F_CALC_SENSOR_POS( N44_AI2_CH5_4 * 0.004, ALARMS.Clear, LS301 );
F_CALC_SENSOR_POS( N44_AI0_CH6_4 * 0.004, ALARMS.Clear, LS303 );
F_CALC_SENSOR_POS( N44_AI4_CH8_4 * 0.004, ALARMS.Clear, LS305 );

F_CALC_SENSOR_KG( P301.Bar, L301 );
F_CALC_SENSOR_KG( P303.Bar, L303 );
F_CALC_SENSOR_KG( P305.Bar, L305 );
F_CALC_SENSOR_KG( P307.Bar, L307 );
F_CALC_SENSOR_KG( P309.Bar, L309 );
F_CALC_SENSOR_KG( P311.Bar, L311 );

(*MF04 - Node44*)
SF402 := N38_DI7_CH8_2;
SF403 := N38_DI6_CH8_4;
SF404 := N44_DI1_CH7_2;
SF405 := N44_DI0_CH7_4;

(*MF05 - Node41*)
F_CALC_SENSOR_BAR( N41_AI3_CH5_2 * 0.004, ALARMS.Clear,  P501 );
F_CALC_SENSOR_BAR( N41_AI2_CH5_4 * 0.004, ALARMS.Clear,  P503 );
F_CALC_SENSOR_BAR( N41_AI1_CH6_2 * 0.004, ALARMS.Clear,  P507 );
F_CALC_SENSOR_BAR( N41_AI0_CH6_4 * 0.004, ALARMS.Clear,  P505 );

(*F_CALC_SENSOR_KG( P501.Bar, L501 );*)
F_CALC_SENSOR_KG( P503.Bar, L503 );
F_CALC_SENSOR_KG( P505.Bar, L505 );
L501_7 := P501.Bar * L501.Cal_K - P507.Bar * L501.Cal_C;

(*MF06 - Node20/47*)
F_CALC_SENSOR_BAR ( N20_AI3_CH5_2 * 0.004, ALARMS.Clear,  P601 );
F_CALC_SENSOR_BAR ( N20_AI2_CH5_4 * 0.004, ALARMS.Clear,  P603 );
F_CALC_SENSOR_BAR ( N20_AI1_CH6_2 * 0.004, ALARMS.Clear,  P605 );
F_CALC_SENSOR_BAR ( N20_AI0_CH6_4 * 0.004, ALARMS.Clear,  P607 );

F_CALC_SENSOR_POS ( N47_AI1_CH6_2 * 0.004, ALARMS.Clear, LS601 );
F_CALC_SENSOR_POS ( N20_AI4_CH8_4 * 0.004, ALARMS.Clear, LS605 );


(*MF07 - Node21/22*)
F_CALC_SENSOR_BAR( N21_AI3_CH5_2 * 0.004, ALARMS.Clear,  P701 );
F_CALC_SENSOR_BAR( N21_AI2_CH5_4 * 0.004, ALARMS.Clear,  P703 );

F_CALC_SENSOR_POS( N21_AI1_CH6_2 * 0.004, ALARMS.Clear, LS707 );
F_CALC_SENSOR_POS( N21_AI0_CH6_4 * 0.004, ALARMS.Clear, LS709 );

F_CALC_SENSOR_BAR( N22_AI3_CH5_2 * 0.004, ALARMS.Clear,  P707 );
F_CALC_SENSOR_BAR( N22_AI2_CH5_4 * 0.004, ALARMS.Clear,  P709 );
F_CALC_SENSOR_BAR( N22_AI1_CH6_2 * 0.004, ALARMS.Clear,  P705 );

F_CALC_SENSOR_KG( P701.Bar, L701 );
F_CALC_SENSOR_KG( P703.Bar, L703 );
F_CALC_SENSOR_KG( P705.Bar, L705 );
F_CALC_SENSOR_KG( P707.Bar, L707 );
F_CALC_SENSOR_KG( P709.Bar, L709 );

(*MF08 - Node23*)
F_CALC_SENSOR_NC ( NOT N39_DI3_CH6_2 , ALARMS.Clear, MAIN.Cycle_Time, 0.0, SF801 );
F_CALC_SENSOR_NC ( NOT N39_DI2_CH6_4 , ALARMS.Clear, MAIN.Cycle_Time, 0.0, SF803 );

F_CALC_SENSOR_BAR( N23_AI1_CH6_2 * 0.004, ALARMS.Clear,  P804 );(**)
F_CALC_SENSOR_BAR( N23_AI0_CH6_4 * 0.004, ALARMS.Clear,  P802 );(**)

F_CALC_SENSOR_POS( N23_AI3_CH5_2 * 0.004, ALARMS.Clear, LS803 );(**)
F_CALC_SENSOR_POS( N23_AI2_CH5_4 * 0.004, ALARMS.Clear, LS801 );(**)

(*MF09 - Node35*)
F_CALC_SENSOR_BAR( N35_AI3_CH5_2 * 0.004, ALARMS.Clear,  P901 );
F_CALC_SENSOR_BAR( N35_AI2_CH5_4 * 0.004, ALARMS.Clear,  P903 );
F_CALC_SENSOR_BAR( N35_AI1_CH6_2 * 0.004, ALARMS.Clear,  P905 );
F_CALC_SENSOR_BAR( N35_AI0_CH6_4 * 0.004, ALARMS.Clear,  P907 );

F_CALC_SENSOR_KG( P901.Bar, L901 );
F_CALC_SENSOR_KG( P903.Bar, L903 );

F_CALC_SENSOR_POS( N38_AI3_CH5_2 * 0.004, ALARMS.Clear, LS901 );
F_CALC_SENSOR_POS( N38_AI2_CH5_4 * 0.004, ALARMS.Clear, LS903 );

(*MF10 - Node39/40*)
F_CALC_SENSOR_NC ( N39_DI1_CH7_2, ALARMS.Clear, MAIN.Cycle_Time, 0.0            , SF1002 );
F_CALC_SENSOR_NC (NOT N40_DI7_CH8_2, ALARMS.Clear, MAIN.Cycle_Time, PARAMS.SF_Delay, SF1003 );
F_CALC_SENSOR_NC (NOT N40_DI6_CH8_4, ALARMS.Clear, MAIN.Cycle_Time, PARAMS.SF_Delay, SF1004 );

F_CALC_SENSOR_BAR( N40_AI3_CH5_2 * 0.004, ALARMS.Clear,  P1001 );
F_CALC_SENSOR_BAR( N40_AI2_CH5_4 * 0.004, ALARMS.Clear,  P1002 );
F_CALC_SENSOR_POS( N40_AI1_CH6_2 * 0.004, ALARMS.Clear, LS1002 );(**)
F_CALC_SENSOR_POS( N40_AI0_CH6_4 * 0.004, ALARMS.Clear, LS1001 );(**)

(*MF11 - Node47*)
F_CALC_SENSOR_BAR( N47_AI3_CH5_2 * 0.004, ALARMS.Clear,  P1101 );
F_CALC_SENSOR_BAR( N47_AI2_CH5_4 * 0.004, ALARMS.Clear,  P1102 );

F_CALC_SENSOR_TEMP( N47_AI4_CH8_4 * 0.001, ALARMS.Clear, MAIN.Cycle_Time, S1100 );

(*MF12 - Node24/25*)
F_CALC_SENSOR_BAR( N24_AI7_CH3_2 * 0.001, ALARMS.Clear,  P1216 );
F_CALC_SENSOR_BAR( N24_AI6_CH3_4 * 0.001, ALARMS.Clear,  P1219 );
F_CALC_SENSOR_BAR( N24_AI3_CH5_2 * 0.001, ALARMS.Clear,  P1214 );
F_CALC_SENSOR_BAR( N24_AI2_CH5_4 * 0.001, ALARMS.Clear,  P1215 );
F_CALC_SENSOR_BAR( N24_AI1_CH6_2 * 0.001, ALARMS.Clear,  P1212 );
F_CALC_SENSOR_BAR( N24_AI0_CH6_4 * 0.001, ALARMS.Clear,  P1213 );
F_CALC_SENSOR_BAR( N24_AI5_CH8_2 * 0.001, ALARMS.Clear,  P1210 );
F_CALC_SENSOR_BAR( N24_AI4_CH8_4 * 0.001, ALARMS.Clear,  P1211 );

F_CALC_SENSOR_BAR( N25_AI7_CH3_2 * 0.001, ALARMS.Clear,  P1208 );
F_CALC_SENSOR_BAR( N25_AI6_CH3_4 * 0.001, ALARMS.Clear,  P1209 );
F_CALC_SENSOR_BAR( N25_AI3_CH5_2 * 0.001, ALARMS.Clear,  P1206 );
F_CALC_SENSOR_BAR( N25_AI2_CH5_4 * 0.001, ALARMS.Clear,  P1207 );
F_CALC_SENSOR_BAR( N25_AI1_CH6_2 * 0.001, ALARMS.Clear,  P1204 );
F_CALC_SENSOR_BAR( N25_AI0_CH6_4 * 0.001, ALARMS.Clear,  P1205 );
F_CALC_SENSOR_BAR( N25_AI5_CH8_2 * 0.001, ALARMS.Clear,  P1202 );
F_CALC_SENSOR_BAR( N25_AI4_CH8_4 * 0.001, ALARMS.Clear,  P1203 );

(*MF13 - Node33 - Traveller*)
SF1301 := N38_DI1_CH7_2;
SF1302 := N38_DI0_CH7_4;

F_CALC_SENSOR_BAR( N33_AI3_CH5_2 * 0.004, ALARMS.Clear,  P1302 );
F_CALC_SENSOR_BAR( N33_AI2_CH5_4 * 0.004, ALARMS.Clear,  P1301 );

F_CALC_SENSOR_POS( N38_AI1_CH6_2 * 0.004, ALARMS.Clear, LS1303 );

(*MF16 - Node34*)
F_CALC_SENSOR_BAR( N34_AI3_CH5_2 * 0.001, ALARMS.Clear,  P1603 );
F_CALC_SENSOR_BAR( N34_AI2_CH5_4 * 0.001, ALARMS.Clear,  P1605 );
F_CALC_SENSOR_BAR( N34_AI1_CH6_2 * 0.001, ALARMS.Clear,  P1604 );
F_CALC_SENSOR_BAR( N34_AI0_CH6_4 * 0.001, ALARMS.Clear,  P1602 );

(*MF19 - Node32*)
F_CALC_SENSOR_POS( N32_AI1_CH6_2 * 0.004, ALARMS.Clear, LS1905 );

SF1909 := N32_DI1_CH7_2;
SF1911 := N32_DI0_CH7_4;
SF1901 := N32_DI7_CH8_2;
SF1903 := N32_DI6_CH8_4;

(*MF20 - Node31*)
F_CALC_SENSOR_POS( N31_AI3_CH5_2 * 0.004, ALARMS.Clear, LS2001 );
F_CALC_SENSOR_POS( N31_AI2_CH5_4 * 0.001, ALARMS.Clear, LS2005 );

SF2009 := N31_DI1_CH7_2;
SF2011 := N31_DI0_CH7_4;

(*MF21 - Node28*)
SF2101 := N28_DI5_CH5_2;
SF2103 := N28_DI4_CH5_4;
SF2105 := N28_DI3_CH6_2;
SF2107 := N28_DI2_CH6_4;
SF2109 := N28_DI1_CH7_2;
SF2111 := N28_DI0_CH7_4;

(*MF22 - Node27*)
SF2205 := N27_DI3_CH6_2;
SF2207 := N27_DI2_CH6_4;
SF2209 := N27_DI1_CH7_2;
SF2211 := N27_DI0_CH7_4;

(*MF23 - Node30*)
F_CALC_SENSOR_POS( N30_AI3_CH5_2 * 0.004, ALARMS.Clear, LS021  );
F_CALC_SENSOR_POS( N30_AI2_CH5_4 * 0.004, ALARMS.Clear, LS022  );
F_CALC_SENSOR_POS( N30_AI1_CH6_2 * 0.004, ALARMS.Clear, LS2301 );
F_CALC_SENSOR_POS( N30_AI0_CH6_4 * 0.004, ALARMS.Clear, LS2305 );

SF2309 := N30_DI1_CH7_2;
SF2311 := N30_DI0_CH7_4;
SF021  := N30_DI7_CH8_2;
SF022  := N30_DI6_CH8_4;

(*MF24 - Node29*)
F_CALC_SENSOR_POS( N29_AI3_CH5_2 * 0.001, ALARMS.Clear, LS2401 );
F_CALC_SENSOR_POS( N29_AI2_CH5_4 * 0.004, ALARMS.Clear, LS2409 );
F_CALC_SENSOR_POS( N29_AI1_CH6_2 * 0.004, ALARMS.Clear, LS2201 );
F_CALC_SENSOR_POS( N29_AI0_CH6_4 * 0.004, ALARMS.Clear, LS023  );

SF2405 := N29_DI1_CH7_2;
SF2407 := N29_DI0_CH7_4;

(*MF25 - Node26*)
F_CALC_SENSOR_POS( N26_AI3_CH5_2 * 0.004, ALARMS.Clear, LS2501 );
F_CALC_SENSOR_POS( N26_AI2_CH5_4 * 0.004, ALARMS.Clear, LS2505 );
F_CALC_SENSOR_BAR( N26_AI1_CH6_2 * 0.004, ALARMS.Clear, P2500  );
F_CALC_SENSOR_POS( N26_AI0_CH6_4 * 0.004, ALARMS.Clear, LS024  );

SF023  := N26_DI7_CH8_2;
SF024  := N26_DI6_CH8_4;


(*DGB Sela - Node48*)
F_CALC_SENSOR_BAR ( N48_AI3_CH5_2 * 0.004, ALARMS.Clear,  P_SealP );
F_CALC_SENSOR_BAR ( N48_AI1_CH6_2 * 0.004, ALARMS.Clear,  P_SealS );


(*L102_raw := P102_bar * PARAMS.stL102_Cal.K;*)

(*L102_Kg := L102_raw * (PARAMS.stL102_Cal.C / 100.0);*)

(*Buttons*)
(*FRO TACK*)
B301[1] := N102_IN.2;
B302[1] := N102_IN.3;
B301[2] := N113_IN.3;
B302[2] := N113_IN.2;
(*A3 TACK*)
B303[1] := N102_IN.4;
B304[1] := N102_IN.5;
B303[2] := N113_IN.5;
B304[2] := N113_IN.4;
(*J5*)
B305[1] := N118_IN.6;
B306[1] := N118_IN.7;
B305[2] := N119_IN.7;
B306[2] := N119_IN.6;
(*J4*)
B307[1] := N118_IN.8;
B308[1] := N118_IN.9;
B307[2] := N119_IN.9;
B308[2] := N119_IN.8;
(*FORESTAY*)
B309[1] := N104_IN.1;
B310[1] := N104_IN.0;
B309[2] := N105_IN.0;
B310[2] := N105_IN.1;
(*J2*)
B311[1] := N114_IN.4;
B312[1] := N114_IN.5;
B311[2] := N115_IN.5;
B312[2] := N115_IN.4;
(*JIB INOUT*)
B501[1] := N114_IN.2;
B502[1] := N114_IN.3;
B501[2] := N115_IN.3;
B502[2] := N115_IN.2;
(*JIB UPDW*)
B503[1] := N114_IN.0;
B504[1] := N114_IN.1;
B503[2] := N115_IN.1;
B504[2] := N115_IN.0;
(*VANG*)
(*B505 [1] := N116_IN.4;
B506 [1] := N116_IN.5;
B506Q[1] := N116_IN.5 AND N116_IN.0;
B505 [2] := N117_IN.5;
B506 [2] := N117_IN.4;
B506Q[2] := N117_IN.4 AND N117_IN.1;*)

(*PORP UP/DW*)
B601[1] := N112_IN.3; (*DW*)
B603[1] := N112_IN.2; (*UP*)
(*TRIM TAB*)
B605[1] := N104_IN.3;
B607[1] := N104_IN.2;
B606[1] := N104_IN.4;
B605[2] := N105_IN.3;
B607[2] := N105_IN.2;
B606[2] := N105_IN.5;

(*INNER STAYSAIL*)
B701[1] := N102_IN.0;
B702[1] := N102_IN.1;
B701[2] := N113_IN.1;
B702[2] := N113_IN.0;
(*MAIN OUTHAUL*)
B703[1] := N116_IN.8;
B704[1] := N116_IN.9;
B703[2] := N117_IN.9;
B704[2] := N117_IN.8;
(*MAIN CUNNINGHAM*)
B705[1] := N116_IN.6;
B706[1] := N116_IN.7;
B705[2] := N117_IN.7;
B706[2] := N117_IN.6;
(*BOTTOM DEFLECTOR*)
B707[1] := N118_IN.2;
B708[1] := N118_IN.3;
B707[2] := N119_IN.3;
B708[2] := N119_IN.2;
(*TOP DEFLECTOR*)
B709[1] := N118_IN.4;
B710[1] := N118_IN.5;
B709[2] := N119_IN.5;
B710[2] := N119_IN.4;

(*BACSTAY PORT*)
(*B901[1] := N104_IN.7; (*Panel Stbd works on Backstay Port*)
B902[1] := N104_IN.6;

B901[2] := N118_IN.0; (*Panel Port works on Backstay Port Fine Tune*)
B902[2] := N118_IN.1;*)

(*BACKSTAY STBD*)
(*B903[1] := N105_IN.6; (*Panel Port works on Backstay Stbd*)
B904[1] := N105_IN.7;

B903[2] := N119_IN.1; (*Panel Stbd works on Backstay Stbd Fine Tune*)
B904[2] := N119_IN.0;*)

(*BACKSTAY TACK*)
(*B90T[1] := N104_IN.5;
B90T[2] := N105_IN.4;*)
(******************************************************fine tune y TACK***)

(*TRAVELLER*)
BTravA[1] := N116_IN.3;
BTravB[1] := N116_IN.2;
BTravT[1] := N116_IN.1;
BTravD[1] := N116_IN.1 AND N116_IN.0;

BTravA[2] := N117_IN.3;
BTravB[2] := N117_IN.2;
BTravT[2] := N117_IN.0;
BTravD[2] := N117_IN.0 AND N117_IN.1;

BTravA[3] := N38_DI0_CH7_4; (******************************Verificar cual es Port y Stbd***)
BTravB[3] := N38_DI1_CH7_2;

(*KEEL*)
BKeelP[1] := N110_IN.0;
BKeelS[1] := N110_IN.4;
BKeelC[1] := N110_IN.3;
BKeelF[1] := N110_IN.2;
BKeelT[1] := N110_IN.5;

BKeelP[2] := N111_IN.0;
BKeelS[2] := N111_IN.4;
BKeelC[2] := N111_IN.3;
BKeelF[2] := N111_IN.2;
BKeelT[2] := N111_IN.5;

(*BKeelP[3] := N108_IN.0;
BKeelS[3] := N108_IN.4;
BKeelC[3] := N108_IN.3;
BKeelF[3] := N108_IN.2;

BKeelP[4] := N109_IN.0;
BKeelS[4] := N109_IN.4;
BKeelC[4] := N109_IN.3;
BKeelF[4] := N109_IN.2;*) (*Now Mast setup*)

(*BOARD*)
BBoardP[1] := MAIN.fbMastSetup.State_MS = 0 AND N108_IN.6;
BBoardS[1] := MAIN.fbMastSetup.State_MS = 0 AND N108_IN.7;
BBoardC[1] := MAIN.fbMastSetup.State_MS = 0 AND N108_IN.5;

BBoardP[2] := MAIN.fbMastSetup.State_HS = 0 AND N109_IN.6;
BBoardS[2] := MAIN.fbMastSetup.State_HS = 0 AND N109_IN.7;
BBoardC[2] := MAIN.fbMastSetup.State_HS = 0 AND N109_IN.5;

(*Bow Thruster*)
BBowThrP := N38_DI7_CH8_2;
BBowThrS := N38_DI6_CH8_4;
BBowThrU := N112_IN.4;
BBowThrD := N112_IN.5;

(*Water Ballast*)
BWB_P_Fwd[1] := N106_IN.0;
BWB_S_Fwd[1] := N106_IN.1;
BWB_P_Aft[1] := N106_IN.2;
BWB_S_Aft[1] := N106_IN.3;
BWB_Fill [1] := N106_IN.4;
BWB_Dump [1] := N106_IN.5;
BWB_Stop [1] := N106_IN.7;
BWB_12   [1] := N106_IN.8;
BWB_Move [1] := N106_IN.9;

BWB_P_Fwd[2] := N107_IN.0;
BWB_S_Fwd[2] := N107_IN.1;
BWB_P_Aft[2] := N107_IN.2;
BWB_S_Aft[2] := N107_IN.3;
BWB_Fill [2] := N107_IN.4;
BWB_Dump [2] := N107_IN.5;
BWB_Stop [2] := N107_IN.7;
BWB_12   [2] := N107_IN.8;
BWB_Move [2] := N107_IN.9;

(*Ligths*)
L_Red_Trig   ( CLK:= N103_IN.0 );
L_Anchor_Trig( CLK:= N103_IN.1 );
L_Steam_Trig ( CLK:= N103_IN.2 );
L_Deck_Trig  ( CLK:= N103_IN.3 );
L_Nav_Trig   ( CLK:= N103_IN.4 );

L_HMI_Red_Trig   ( );
L_HMI_Anchor_Trig( );
L_HMI_Steam_Trig ( );
L_HMI_Deck_Trig  ( );
L_HMI_Nav_Trig   ( );

L_Red    := L_Red_Trig.CLK    OR L_HMI_Red_Trig.CLK;
L_Anchor := L_Anchor_Trig.CLK OR L_HMI_Anchor_Trig.CLK;
L_Steam  := L_Steam_Trig.CLK  OR L_HMI_Steam_Trig.CLK;
L_Deck   := L_Deck_Trig.CLK   OR L_HMI_Deck_Trig.CLK;
L_Nav    := L_Nav_Trig.CLK    OR L_HMI_Nav_Trig.CLK;

Override_Trig( CLK:= N117_IN.1 );
RemPort_Trig ( CLK:= N105_IN.4 );
RemStbd_Trig ( CLK:= N104_IN.5 );
RemOff_Trig  ( CLK:= N20_DI0 OR N20_DI1 OR N20_DI3 OR N20_DI4);

IF Override_Trig.Q THEN
	Override_ON := NOT Override_ON;
END_IF

IF RemPort_Trig.Q THEN
	RemPort_ON := NOT RemPort_ON;
END_IF

IF RemStbd_Trig.Q THEN
	RemStbd_ON := NOT RemStbd_ON;
END_IF

IF RemOff_Trig.Q THEN
	RemPort_ON := FALSE;
	RemStbd_ON := FALSE;
END_IF

(*W1202 - Prim Stbd*)
IF NOT RemStbd_ON THEN
	B1202_1[1] := N10_DI0;
	B1202_2[1] := N10_DI1;
ELSE
	B1202_1[1] := FALSE;
	B1202_2[1] := FALSE;
END_IF

B1202_G    := N10_DI2;
B1202_1[4] := N120_IN.3;
B1202_2[4] := N120_IN.8;

(* W1204 - Pit Stbd*)
B1204_1[1] := N10_DI6;
B1204_2[1] := N10_DI7;
B1204_G    := FALSE;
B1204_1[4] := N120_IN.1;
B1204_2[4] := N120_IN.6;

(*W1206 - MAIN*)
B1206_1[1] := N20_DI0;
B1206_2[1] := N20_DI1;
B1206_G    := N20_DI2;
B1206_1[2] := N20_DI3;
B1206_2[2] := N20_DI4;
B1206_1[4] := N120_IN.0;
B1206_2[4] := N120_IN.5;

IF RemStbd_ON AND RemPOrt_ON THEN
	B1206_1[3] := N10_DI0 OR N11_DI0;
	B1206_2[3] := N10_DI1 OR N11_DI1;
ELSIF RemStbd_ON THEN
	B1206_1[3] := N10_DI0;
	B1206_2[3] := N10_DI1;
ELSIF RemPort_ON THEN
	B1206_1[3] := N11_DI0;
	B1206_2[3] := N11_DI1;
ELSE
	B1206_1[3] := FALSE;
	B1206_2[3] := FALSE;
END_IF

(*W1208 - Runn Port*)
B1208_1[1] := N13_DI0;
B1208_2[1] := N13_DI1;
B1208_G    := N13_DI2;
B1208_1[4] := N121_IN.0;
B1208_2[4] := N121_IN.4;

(*W1210 - Prim Port*)
IF NOT RemPort_ON THEN
	B1210_1[1] := N11_DI0;
	B1210_2[1] := N11_DI1;
ELSE
	B1210_1[1] := FALSE;
	B1210_2[1] := FALSE;
END_IF

B1210_G    := N11_DI2;
B1210_1[4] := N121_IN.1;
B1210_2[4] := N121_IN.5;

(*W1212 - Sec Port*)
B1212_1[1] := N11_DI3;
B1212_2[1] := N11_DI4;
B1212_G    := N11_DI5;
B1212_1[4] := N121_IN.2;
B1212_2[4] := N121_IN.6;

(* W1214 - Pit Port*)
B1214_1[1] := N11_DI6;
B1214_2[1] := N11_DI7;
B1214_G    := FALSE;
B1214_1[4] := N121_IN.3;
B1214_2[4] := N121_IN.7;

(*W1602 - Runn Stbd*)
B1602_1[1] := N12_DI0;
B1602_2[1] := N12_DI1;
B1602_G    := N12_DI2;
B1602_1[4] := N120_IN.4;
B1602_2[4] := N120_IN.9;

(*W1604 - Sec Stbd*)
B1604_1[1] := N10_DI3;
B1604_2[1] := N10_DI4;
B1604_G    := N10_DI5;
B1604_1[4] := N120_IN.2;
B1604_2[4] := N120_IN.7;

(*****************)
(* CAN NODESTATE *)
(*****************)
F_CALC_CAN_STATE ( CAN1_State, ALARMS.Clear,  CAN1 );
F_CALC_CAN_STATE ( CAN2_State, ALARMS.Clear,  CAN2 );
F_CALC_CAN_STATE ( CAN3_State, ALARMS.Clear,  CAN3 );
F_CALC_CAN_STATE ( CAN4_State, ALARMS.Clear,  CAN4 );
F_CALC_CAN_STATE ( CAN5_State, ALARMS.Clear,  CAN5 );

F_CALC_CAN_NODESTATE( J1939_NodeState, ALARMS.Clear, NJ1939 );

F_CALC_CAN_NODESTATE ( N20_NodeState, ALARMS.Clear,  N20 );
F_CALC_CAN_NODESTATE ( N21_NodeState, ALARMS.Clear,  N21 );
F_CALC_CAN_NODESTATE ( N22_NodeState, ALARMS.Clear,  N22 );
F_CALC_CAN_NODESTATE ( N23_NodeState, ALARMS.Clear,  N23 );
F_CALC_CAN_NODESTATE ( N24_NodeState, ALARMS.Clear,  N24 );
F_CALC_CAN_NODESTATE ( N25_NodeState, ALARMS.Clear,  N25 );
F_CALC_CAN_NODESTATE ( N26_NodeState, ALARMS.Clear,  N26 );
F_CALC_CAN_NODESTATE ( N27_NodeState, ALARMS.Clear,  N27 );
F_CALC_CAN_NODESTATE ( N28_NodeState, ALARMS.Clear,  N28 );
F_CALC_CAN_NODESTATE ( N29_NodeState, ALARMS.Clear,  N29 );
F_CALC_CAN_NODESTATE ( N30_NodeState, ALARMS.Clear,  N30 );
F_CALC_CAN_NODESTATE ( N31_NodeState, ALARMS.Clear,  N31 );
F_CALC_CAN_NODESTATE ( N32_NodeState, ALARMS.Clear,  N32 );
F_CALC_CAN_NODESTATE ( N33_NodeState, ALARMS.Clear,  N33 );
F_CALC_CAN_NODESTATE ( N34_NodeState, ALARMS.Clear,  N34 );
F_CALC_CAN_NODESTATE ( N35_NodeState, ALARMS.Clear,  N35 );
F_CALC_CAN_NODESTATE ( N36_NodeState, ALARMS.Clear,  N36 );
F_CALC_CAN_NODESTATE ( N37_NodeState, ALARMS.Clear,  N37 );
F_CALC_CAN_NODESTATE ( N38_NodeState, ALARMS.Clear,  N38 );
F_CALC_CAN_NODESTATE ( N39_NodeState, ALARMS.Clear,  N39 );
F_CALC_CAN_NODESTATE ( N40_NodeState, ALARMS.Clear,  N40 );
F_CALC_CAN_NODESTATE ( N41_NodeState, ALARMS.Clear,  N41 );
F_CALC_CAN_NODESTATE ( N42_NodeState, ALARMS.Clear,  N42 );
F_CALC_CAN_NODESTATE ( N43_NodeState, ALARMS.Clear,  N43 );
F_CALC_CAN_NODESTATE ( N44_NodeState, ALARMS.Clear,  N44 );
F_CALC_CAN_NODESTATE ( N47_NodeState, ALARMS.Clear,  N47 );

F_CALC_CAN_NODESTATE ( N50_NodeState, ALARMS.Clear,  N50 );
F_CALC_CAN_NODESTATE ( N51_NodeState, ALARMS.Clear,  N51 );
F_CALC_CAN_NODESTATE ( N52_NodeState, ALARMS.Clear,  N52 );
F_CALC_CAN_NODESTATE ( N53_NodeState, ALARMS.Clear,  N53 );
F_CALC_CAN_NODESTATE ( N54_NodeState, ALARMS.Clear,  N54 );
F_CALC_CAN_NODESTATE ( N55_NodeState, ALARMS.Clear,  N55 );
F_CALC_CAN_NODESTATE ( N56_NodeState, ALARMS.Clear,  N56 );
F_CALC_CAN_NODESTATE ( N57_NodeState, ALARMS.Clear,  N57 );
F_CALC_CAN_NODESTATE ( N58_NodeState, ALARMS.Clear,  N58 );
F_CALC_CAN_NODESTATE ( N59_NodeState, ALARMS.Clear,  N59 );
F_CALC_CAN_NODESTATE ( N60_NodeState, ALARMS.Clear,  N60 );
F_CALC_CAN_NODESTATE ( N61_NodeState, ALARMS.Clear,  N61 );
F_CALC_CAN_NODESTATE ( N64_NodeState, ALARMS.Clear,  N64 );
F_CALC_CAN_NODESTATE ( N70_NodeState, ALARMS.Clear,  N70 );
F_CALC_CAN_NODESTATE ( N71_NodeState, ALARMS.Clear,  N71 );
F_CALC_CAN_NODESTATE ( N72_NodeState, ALARMS.Clear,  N72 );
F_CALC_CAN_NODESTATE ( N73_NodeState, ALARMS.Clear,  N73 );
F_CALC_CAN_NODESTATE ( N74_NodeState, ALARMS.Clear,  N74 );

F_CALC_CAN_NODESTATE ( N102_NodeState, ALARMS.Clear,  N102 );
F_CALC_CAN_NODESTATE ( N103_NodeState, ALARMS.Clear,  N103 );
F_CALC_CAN_NODESTATE ( N104_NodeState, ALARMS.Clear,  N104 );
F_CALC_CAN_NODESTATE ( N105_NodeState, ALARMS.Clear,  N105 );
F_CALC_CAN_NODESTATE ( N106_NodeState, ALARMS.Clear,  N106 );
F_CALC_CAN_NODESTATE ( N107_NodeState, ALARMS.Clear,  N107 );
F_CALC_CAN_NODESTATE ( N108_NodeState, ALARMS.Clear,  N108 );
F_CALC_CAN_NODESTATE ( N109_NodeState, ALARMS.Clear,  N109 );
F_CALC_CAN_NODESTATE ( N110_NodeState, ALARMS.Clear,  N110 );
F_CALC_CAN_NODESTATE ( N111_NodeState, ALARMS.Clear,  N111 );
F_CALC_CAN_NODESTATE ( N112_NodeState, ALARMS.Clear,  N112 );
F_CALC_CAN_NODESTATE ( N113_NodeState, ALARMS.Clear,  N113 );
F_CALC_CAN_NODESTATE ( N114_NodeState, ALARMS.Clear,  N114 );
F_CALC_CAN_NODESTATE ( N115_NodeState, ALARMS.Clear,  N115 );
F_CALC_CAN_NODESTATE ( N116_NodeState, ALARMS.Clear,  N116 );
F_CALC_CAN_NODESTATE ( N117_NodeState, ALARMS.Clear,  N117 );
F_CALC_CAN_NODESTATE ( N118_NodeState, ALARMS.Clear,  N118 );
F_CALC_CAN_NODESTATE ( N119_NodeState, ALARMS.Clear,  N119 );

F_CALC_CAN_NODESTATE ( N10_NodeState, ALARMS.Clear,  N10 );
F_CALC_CAN_NODESTATE ( N11_NodeState, ALARMS.Clear,  N11 );
F_CALC_CAN_NODESTATE ( N12_NodeState, ALARMS.Clear,  N12 );
F_CALC_CAN_NODESTATE ( N13_NodeState, ALARMS.Clear,  N13 );
F_CALC_CAN_NODESTATE ( N20_2_NodeState, ALARMS.Clear,  N20_2 );


(***************)
(* System Time *)
(***************)
fbLocalTime( bEnable := TRUE );

(*
tsTime  := fbLocalTime.systemTime;
sDate   := DWORD_TO_STRING( tsTime.wYear * 10000 + tsTime.wMonth * 100 + tsTime.wDay );
sLocal  := REAL_TO_STRING ( tsTime.wHour * 10000.0 + tsTime.wMinute * 100.0 + tsTime.wSecond + tsTime.wMilliseconds / 1000.0 );
sDaySec := REAL_TO_STRING ( tsTime.wHour * 3600.0  + tsTime.wMinute * 60.0  + tsTime.wSecond + tsTime.wMilliseconds / 1000.0 );
*)

sLocal    := SYSTEMTIME_TO_STRING(fbLocalTime.systemTime); (*YYYY-MM-DD-hh:mm:ss.sss*)
sLocal    := DELETE (sLocal, 11, 1); (*hh:mm:ss.sss*)
sVisuTime := DELETE (sLocal,  4, 9); (*hh:mm:ss*)
END_PROGRAM

(* POU PARAMS, ST *)
PROGRAM PARAMS
VAR CONSTANT
	BUF_SIZE: WORD := 15000;
END_VAR
VAR
	Loaded : BOOL;
	Error  : BOOL;
	Save   : BOOL;
	Saved  : BOOL;
	State  : WORD;
	SavedCnt : REAL;

	fbParamList : FB_IDLIST;
	fbSaveList  : FB_FILE_WRITE;

	aBuffer : ARRAY[1..BUF_SIZE] OF BYTE;
	wBufPos : DWORD;

	i : INT;

(*Sensors*)
	SF_Delay : REAL;

(*Parameters*)
	(*stTankCfg*)
	stEngineCfg     : ST_ENGINE_CFG;
	stPropulsionCfg : ST_PROPULSION_CFG;
	stPowerpackCfg  : ST_POWERPACK_CFG;

	(*Cilinders*)
	stSE301Cfg  : ST_SE_CYLINDER_POS_CFG;
	stSE303Cfg  : ST_SE_CYLINDER_POS_CFG;
	stSE305Cfg  : ST_SE_CYLINDER_POS_CFG;
	stSE307Cfg  : ST_SE_CYLINDER_POS_CFG;
	stSE309Cfg  : ST_SE_CYLINDER_POS_CFG;
	stSE311Cfg  : ST_SE_CYLINDER_POS_CFG;

	stSE501Cfg  : ST_SE_CYLINDER_CFG;
	stSE503Cfg  : ST_SE_CYLINDER_CFG;
	stSE505Cfg  : ST_SE_CYLINDER_CFG;

	stDE601Cfg  : ST_LIFT_PROP_CFG;
	stDE605Cfg  : ST_DE_CYLINDER_POS_CFG;

	stSE701Cfg  : ST_SE_CYLINDER_CFG;
	stSE703Cfg  : ST_SE_CYLINDER_CFG;
	stSE705Cfg  : ST_SE_CYLINDER_CFG;
	stSE707Cfg  : ST_SE_CYLINDER_POS_CFG;
	stSE709Cfg  : ST_SE_CYLINDER_POS_CFG;

	stSE901Cfg  : ST_SE_CYLINDER_POS_CFG;
	(*stSE903Cfg  : ST_SE_CYLINDER_POS_CFG;*)

	(*Water Ballast*)
	stWBCfg        : ST_WB_CFG;
	stWBValveSFCfg : ST_WB_VALVE_CFG;
	stWBValveLSCfg : ST_WB_VALVE_LS_CFG;

	(*Winches*)
	stW1202Cfg    : ST_WINCHE_CFG;
	stW1204Cfg    : ST_WINCHE_CFG;
	stW1206Cfg    : ST_WINCHE_CFG;
	stW1208Cfg    : ST_WINCHE_CFG;
	stW1210Cfg    : ST_WINCHE_CFG;
	stW1212Cfg    : ST_WINCHE_CFG;
	stW1214Cfg    : ST_WINCHE_CFG;

	stW1602Cfg    : ST_WINCHE_CFG;
	stW1604Cfg    : ST_WINCHE_CFG;

	stWRampCfg    : ST_WINCHE_RAMP_CFG;

	(*Other*)
	stBoardCfg     : ST_BOARD_CFG;
	stKeelCfg      : ST_KEEL_CFG;
	stTravellerCfg : ST_TRAVELLER_CFG;

	stBowThrCfg     : ST_LP_FUNC_CFG;
	stBowThrUpDwCfg : ST_LP_FUNC_CFG;

	stTackValveCfg  : ST_TACK_VALVE_CFG;

	stMastSetup : ST_MAST_SETUP;

(*UDP Parameter Vars*)
	sUDPSendHost : STRING(15);
	nUDPSendPort : UDINT;
	nUDPSendTime : UINT;
	nUDPRecvPort : UDINT;

	sUDPAlarmsHost : STRING(15);
	nUDPAlarmsPort : UDINT;
END_VAR
IF SavedCnt > 0 THEN
	Saved    := FALSE;
	SavedCnt := SavedCnt - 0.005;
ELSE
	Saved := TRUE;
END_IF

CASE State OF
0: (*Init State*)
	IF NOT Loaded THEN
		fbParamList.sFilePath := '\Hard Disk\FTP\Sensors.txt';
		(*fbParamList.sFilePath := '\Hard Disk\FTP\Parameters.txt';*)
		Error := FALSE;
		State := 100;
	ELSIF Save THEN
		fbSaveList.sFilePath := '\Hard Disk\FTP\';
		fbSaveList.sFileName := 'Sensors';
(*		fbSaveList.sFileName := 'Parameters';*)
		fbSaveList.sFileExt  := '.txt';
		fbSaveList.Backup    := TRUE;

		Save  := FALSE;
		SavedCnt := 1.5;
		State := 200;
	ELSE
		fbParamList( bEnable := FALSE );
		fbSaveList ( bEnable := FALSE );

	END_IF

100: (*Load Sensors*)
	fbParamList( bEnable := TRUE );

	IF fbParamList.bInit THEN
		State := 110;
	ELSIF fbParamList.byError > 0 THEN
		Loaded := TRUE;
		Error  := TRUE;
		State  := 0;
	END_IF

110:(*Read SENSORS*)
	(*EVP*)
	EVP313.Cal_K    := F_IDLIST_GETREAL( 'EVP313_K'   , fbParamList );
	EVP313.Cal_Off  := F_IDLIST_GETREAL( 'EVP313_Off' , fbParamList );
	EVP513.Cal_K    := F_IDLIST_GETREAL( 'EVP513_K'   , fbParamList );
	EVP513.Cal_Off  := F_IDLIST_GETREAL( 'EVP513_Off' , fbParamList );
	EVP709.Cal_K    := F_IDLIST_GETREAL( 'EVP709_K'   , fbParamList );
	EVP709.Cal_Off  := F_IDLIST_GETREAL( 'EVP709_Off' , fbParamList );
	EVP1005.Cal_K   := F_IDLIST_GETREAL( 'EVP1005_K'  , fbParamList );
	EVP1005.Cal_Off := F_IDLIST_GETREAL( 'EVP1005_Off', fbParamList );
	EVP1010.Cal_K   := F_IDLIST_GETREAL( 'EVP1010_K'  , fbParamList );
	EVP1010.Cal_Off := F_IDLIST_GETREAL( 'EVP1010_Off', fbParamList );

	(*Node36/37 - TANK + GS + MF00 + PP*)
	SF_Delay := F_IDLIST_GETREAL( 'SF_Delay', fbParamList );

	F_READ_SENSOR_BAR(  P010, fbParamList );
	P010.MinBar := F_IDLIST_GETREAL( CONCAT(P010.Name, '_Min'), fbParamList );

	F_READ_SENSOR_BAR(  P001, fbParamList );
	F_READ_SENSOR_BAR(  P002, fbParamList );
	F_READ_SENSOR_BAR(  P003, fbParamList );

	F_READ_SENSOR_BAR(  P051, fbParamList );
	F_READ_SENSOR_BAR(  P052, fbParamList );

	F_READ_SENSOR_TEMP( S011, fbParamList );
	F_READ_SENSOR_TEMP( S100, fbParamList );
	F_READ_SENSOR_TEMP( S101, fbParamList );
	F_READ_SENSOR_TEMP( S102, fbParamList );

	(*Water Ballast - Nodes...*)
	F_READ_SENSOR_POS( LS021, fbParamList );
	F_READ_SENSOR_POS( LS022, fbParamList );
	F_READ_SENSOR_POS( LS023, fbParamList );
	F_READ_SENSOR_POS( LS024, fbParamList );

	(*MF01 - Node42*)
	F_READ_SENSOR_BAR(  P101, fbParamList );
	F_READ_SENSOR_BAR(  P103, fbParamList );

	(*MF02 - Node34*)
	F_READ_SENSOR_BAR(  P201 , fbParamList );

	(*MF03 - Node43/44*)
	F_READ_SENSOR_BAR(  P301, fbParamList );
	F_READ_SENSOR_BAR(  P303, fbParamList );
	F_READ_SENSOR_BAR(  P305, fbParamList );
	F_READ_SENSOR_BAR(  P307, fbParamList );
	F_READ_SENSOR_BAR(  P309, fbParamList );
	F_READ_SENSOR_BAR(  P311, fbParamList );

	F_READ_SENSOR_POS( LS301, fbParamList );
	F_READ_SENSOR_POS( LS303, fbParamList );
	F_READ_SENSOR_POS( LS305, fbParamList );
	F_READ_SENSOR_POS( LS307, fbParamList );
	F_READ_SENSOR_POS( LS309, fbParamList );
	F_READ_SENSOR_POS( LS311, fbParamList );

	F_READ_SENSOR_KG(  L301, fbParamList );
	F_READ_SENSOR_KG(  L303, fbParamList );
	F_READ_SENSOR_KG(  L305, fbParamList );
	F_READ_SENSOR_KG(  L307, fbParamList );
	F_READ_SENSOR_KG(  L309, fbParamList );
	F_READ_SENSOR_KG(  L311, fbParamList );

	(*MF05 - Node41*)
	F_READ_SENSOR_BAR(  P501, fbParamList );
	F_READ_SENSOR_BAR(  P503, fbParamList );
	F_READ_SENSOR_BAR(  P505, fbParamList );
	F_READ_SENSOR_BAR(  P507, fbParamList );

	F_READ_SENSOR_KG(  L501, fbParamList );
	F_READ_SENSOR_KG(  L503, fbParamList );
	F_READ_SENSOR_KG(  L505, fbParamList );

	(*MF06 - Node20*)
	F_READ_SENSOR_BAR(  P601, fbParamList );
	F_READ_SENSOR_BAR(  P603, fbParamList );
	F_READ_SENSOR_BAR(  P605, fbParamList );
	F_READ_SENSOR_BAR(  P607, fbParamList );

	F_READ_SENSOR_POS( LS601, fbParamList );
	F_READ_SENSOR_POS( LS605, fbParamList );

	(*MF07 - Node21/22*)
	F_READ_SENSOR_BAR(  P701, fbParamList );
	F_READ_SENSOR_BAR(  P703, fbParamList );
	F_READ_SENSOR_BAR(  P705, fbParamList );
	F_READ_SENSOR_BAR(  P707, fbParamList );
	F_READ_SENSOR_BAR(  P709, fbParamList );

	F_READ_SENSOR_KG(  L701, fbParamList );
	F_READ_SENSOR_KG(  L703, fbParamList );
	F_READ_SENSOR_KG(  L705, fbParamList );
	F_READ_SENSOR_KG(  L707, fbParamList );
	F_READ_SENSOR_KG(  L709, fbParamList );

	F_READ_SENSOR_POS( LS707, fbParamList );
	F_READ_SENSOR_POS( LS709, fbParamList );

	(*MF08 - Node23*)
	F_READ_SENSOR_BAR(  P802, fbParamList );
	F_READ_SENSOR_BAR(  P804, fbParamList );

	F_READ_SENSOR_POS( LS801, fbParamList );
	F_READ_SENSOR_POS( LS803, fbParamList );

	(*MF09 - Node35*)
	F_READ_SENSOR_BAR(  P901, fbParamList );
	F_READ_SENSOR_BAR(  P903, fbParamList );

	F_READ_SENSOR_KG(  L901, fbParamList );
	F_READ_SENSOR_KG(  L903, fbParamList );

	F_READ_SENSOR_POS( LS901, fbParamList );
	F_READ_SENSOR_POS( LS903, fbParamList );

	(*MF10 - Node40*)
	F_READ_SENSOR_BAR(  P1001, fbParamList );
	F_READ_SENSOR_BAR(  P1002, fbParamList );

	F_READ_SENSOR_POS( LS1001, fbParamList );
	F_READ_SENSOR_POS( LS1002, fbParamList );

	(*MF11 - Node21*)
	F_READ_SENSOR_BAR(  P1101, fbParamList );
	F_READ_SENSOR_BAR(  P1102, fbParamList );
	F_READ_SENSOR_TEMP( S1100, fbParamList );

	(*MF12 - Node24/25*)
	F_READ_SENSOR_BAR(  P1202, fbParamList );
	F_READ_SENSOR_BAR(  P1203, fbParamList );
	F_READ_SENSOR_BAR(  P1204, fbParamList );
	F_READ_SENSOR_BAR(  P1205, fbParamList );
	F_READ_SENSOR_BAR(  P1206, fbParamList );
	F_READ_SENSOR_BAR(  P1207, fbParamList );
	F_READ_SENSOR_BAR(  P1208, fbParamList );
	F_READ_SENSOR_BAR(  P1209, fbParamList );
	F_READ_SENSOR_BAR(  P1210, fbParamList );
	F_READ_SENSOR_BAR(  P1211, fbParamList );
	F_READ_SENSOR_BAR(  P1212, fbParamList );
	F_READ_SENSOR_BAR(  P1213, fbParamList );
	F_READ_SENSOR_BAR(  P1214, fbParamList );
	F_READ_SENSOR_BAR(  P1215, fbParamList );
	F_READ_SENSOR_BAR(  P1216, fbParamList );
	F_READ_SENSOR_BAR(  P1219, fbParamList );

	(*MF13 - Node33 - Traveller*)
	F_READ_SENSOR_BAR(  P1301, fbParamList );
	F_READ_SENSOR_BAR(  P1302, fbParamList );

	F_READ_SENSOR_POS( LS1303, fbParamList );

	(*MF16 - Node34*)
	F_READ_SENSOR_BAR(  P1602, fbParamList );
	F_READ_SENSOR_BAR(  P1603, fbParamList );
	F_READ_SENSOR_BAR(  P1604, fbParamList );
	F_READ_SENSOR_BAR(  P1605, fbParamList );

	(*MF19 - Node32*)
	F_READ_SENSOR_POS( LS1905, fbParamList );

	(*MF20 - Node31*)
	F_READ_SENSOR_POS( LS2001, fbParamList );
	F_READ_SENSOR_POS( LS2005, fbParamList );

	(*MF22 - Node31*)
	F_READ_SENSOR_POS( LS2201, fbParamList );

	(*MF23 - Node30*)
	F_READ_SENSOR_POS( LS2301, fbParamList );
	F_READ_SENSOR_POS( LS2305, fbParamList );

	(*MF24 - Node29*)
	F_READ_SENSOR_POS( LS2401, fbParamList );
	F_READ_SENSOR_POS( LS2409, fbParamList );

	(*MF25 - Node26*)
	F_READ_SENSOR_BAR(  P2500, fbParamList );
	F_READ_SENSOR_POS( LS2501, fbParamList );
	F_READ_SENSOR_POS( LS2505, fbParamList );

	(*DGB Seal - Node48*)
	F_READ_SENSOR_BAR(  P_SealP, fbParamList );
	F_READ_SENSOR_BAR(  P_SealS, fbParamList );


	(*Next State*)
	fbParamList( bEnable := FALSE );
	fbParamList.sFilePath := '\Hard Disk\FTP\Parameters.txt';
	State := 120;

120: (*Load Parameters*)
	fbParamList( bEnable := TRUE );
	IF fbParamList.bInit THEN
		State := 130;
	ELSIF fbParamList.byError > 0 THEN
		Loaded := TRUE;
		Error  := TRUE;
		State  := 0;
	END_IF

130:(*Read PARAMETERS*)

(*1- Engine*)
	F_READ_ENGINE_CFG    ( 'Engine'    , MAIN.Cycle_Time, stEngineCfg    , fbParamList );
	F_READ_POWERPACK_CFG ( 'Powerpack' , MAIN.Cycle_Time, stPowerpackCfg , fbParamList );
	F_READ_PROPULSION_CFG( 'Propulsion', MAIN.Cycle_Time, stPropulsionCfg, fbParamList );


(*2- HP functions*)
	F_READ_SE_CYLINDER_POS_CFG	( 'A3Tack', MAIN.Cycle_Time, stSE301Cfg , fbParamList );
	F_READ_SE_CYLINDER_POS_CFG	( 'FrTack', MAIN.Cycle_Time, stSE303Cfg , fbParamList );
	F_READ_SE_CYLINDER_POS_CFG	( 'J5'    , MAIN.Cycle_Time, stSE305Cfg , fbParamList );
	F_READ_SE_CYLINDER_POS_CFG	( 'J4'    , MAIN.Cycle_Time, stSE307Cfg , fbParamList );
	F_READ_SE_CYLINDER_POS_CFG	( 'Fsy'   , MAIN.Cycle_Time, stSE309Cfg , fbParamList );
	F_READ_SE_CYLINDER_POS_CFG	( 'J2'    , MAIN.Cycle_Time, stSE311Cfg , fbParamList );

	F_READ_SE_CYLINDER_CFG		( 'JibIO' , MAIN.Cycle_Time, stSE501Cfg , fbParamList );
	F_READ_SE_CYLINDER_CFG		( 'JibUD' , MAIN.Cycle_Time, stSE503Cfg , fbParamList );
	F_READ_SE_CYLINDER_CFG		( 'Vang'  , MAIN.Cycle_Time, stSE505Cfg , fbParamList );

	F_READ_LIFT_PROP_CFG        ( 'PropUpDw', MAIN.Cycle_Time, stDE601Cfg, fbParamList );
	F_READ_DE_CYLINDER_POS_CFG	( 'TrimTab' , MAIN.Cycle_Time, stDE605Cfg, fbParamList );

	F_READ_SE_CYLINDER_CFG		( 'Inn'   , MAIN.Cycle_Time, stSE701Cfg , fbParamList );
	F_READ_SE_CYLINDER_CFG		( 'Out'   , MAIN.Cycle_Time, stSE703Cfg , fbParamList );
	F_READ_SE_CYLINDER_CFG		( 'Cunn'  , MAIN.Cycle_Time, stSE705Cfg , fbParamList );
	F_READ_SE_CYLINDER_POS_CFG	( 'Runn'  , MAIN.Cycle_Time, stSE707Cfg , fbParamList );
	F_READ_SE_CYLINDER_POS_CFG	( 'Chksy' , MAIN.Cycle_Time, stSE709Cfg , fbParamList );

	F_READ_SE_CYLINDER_POS_CFG	( 'BsyP'  , MAIN.Cycle_Time, stSE901Cfg , fbParamList );
	(*F_READ_SE_CYLINDER_POS_CFG	( 'BsyS'  , MAIN.Cycle_Time, stSE903Cfg , fbParamList );*)

(*3- Water Ballast*)
	F_READ_WB_CFG        ( 'WB'        , MAIN.Cycle_Time, stWBCfg        , fbParamList );
	F_READ_WB_VALVESF_CFG( 'WBValves'  , MAIN.Cycle_Time, stWBValveSFCfg , fbParamList );
	F_READ_WB_VALVELS_CFG( 'WBValvesLS', MAIN.Cycle_Time, stWBValveLSCfg , fbParamList );

(*4- LP Fucntions*)
	F_READ_WINCHE_CFG ( 'W1202', MAIN.Cycle_Time, stW1202Cfg, fbParamList );
	F_READ_WINCHE_CFG ( 'W1204', MAIN.Cycle_Time, stW1204Cfg, fbParamList );
	F_READ_WINCHE_CFG ( 'W1206', MAIN.Cycle_Time, stW1206Cfg, fbParamList );
	F_READ_WINCHE_CFG ( 'W1208', MAIN.Cycle_Time, stW1208Cfg, fbParamList );
	F_READ_WINCHE_CFG ( 'W1210', MAIN.Cycle_Time, stW1210Cfg, fbParamList );
	F_READ_WINCHE_CFG ( 'W1212', MAIN.Cycle_Time, stW1212Cfg, fbParamList );
	F_READ_WINCHE_CFG ( 'W1214', MAIN.Cycle_Time, stW1214Cfg, fbParamList );
	F_READ_WINCHE_CFG ( 'W1602', MAIN.Cycle_Time, stW1602Cfg, fbParamList );
	F_READ_WINCHE_CFG ( 'W1604', MAIN.Cycle_Time, stW1604Cfg, fbParamList );

	stWRampCfg.Spd_Min := F_IDLIST_GETREAL( 'WRAMP_Min', fbParamList );
	stWRampCfg.Spd_Inc := F_IDLIST_GETREAL( 'WRAMP_Inc', fbParamList );
	stWRampCfg.Spd_Dec := F_IDLIST_GETREAL( 'WRAMP_Dec', fbParamList );

	F_READ_BOARD_CFG    ( 'Board'    , MAIN.Cycle_Time, stBoardCfg    , fbParamList );
	F_READ_KEEL_CFG     ( 'Keel'     , MAIN.Cycle_Time, stKeelCfg     , fbParamList );
	F_READ_TRAVELLER_CFG( 'Traveller', MAIN.Cycle_Time, stTravellerCfg, fbParamList );

	F_READ_LP_FUNC_CFG( 'BowThr'    , MAIN.Cycle_Time, stBowThrCfg    , fbParamList );
	F_READ_LP_FUNC_CFG( 'BowThrUpDw', MAIN.Cycle_Time, stBowThrUpDwCfg, fbParamList );

	F_READ_TACK_VALVE_CFG ('TackValve', MAIN.Cycle_Time, stTackValveCfg, fbParamList );

	F_READ_MAST_SETUP_CFG ('MastSetup', MAIN.Cycle_Time, stMastSetup, fbParamList);

(*UDP Parameter*)
	sUDPSendHost := F_IDLIST_GETSTRING( 'UDPHost', fbParamList );
	nUDPSendPort := F_IDLIST_GETUDINT ( 'UDPPort', fbParamList );
	nUDPSendTime := F_IDLIST_GETUINT  ( 'UDPTime', fbParamList );
    nUDPRecvPort := F_IDLIST_GETUDINT ( 'UDPRecvPort', fbParamList );

	sUDPAlarmsHost := F_IDLIST_GETSTRING( 'UDPAlarmsHost', fbParamList );
	nUDPAlarmsPort := F_IDLIST_GETUDINT ( 'UDPAlarmsPort', fbParamList );

	(*Next State*)
	State := 300;

200: (*Create Sensors Buffer*)
	wBufPos := 0;

(*Sensors*)
	(*EVP PRESS VAR*)
	F_ADD_STRING_TO_BUFFER( S1:= '$n#EVP MAX PRESS VALVE:$n', wSize := BUF_SIZE, pBuffer := ADR(aBuffer), wPos := wBufPos );
	F_ADD_STRINGX4_TO_BUFFER( S1:= 'EVP313_K'   , S2:='$t', S3:= REAL_TO_STRING( EVP313.Cal_K    ), S4:='$n', wSize := BUF_SIZE, pBuffer := ADR(aBuffer), wPos := wBufPos );
	F_ADD_STRINGX4_TO_BUFFER( S1:= 'EVP313_Off' , S2:='$t', S3:= REAL_TO_STRING( EVP313.Cal_Off  ), S4:='$n', wSize := BUF_SIZE, pBuffer := ADR(aBuffer), wPos := wBufPos );
	F_ADD_STRINGX4_TO_BUFFER( S1:= 'EVP513_K'   , S2:='$t', S3:= REAL_TO_STRING( EVP513.Cal_K    ), S4:='$n', wSize := BUF_SIZE, pBuffer := ADR(aBuffer), wPos := wBufPos );
	F_ADD_STRINGX4_TO_BUFFER( S1:= 'EVP513_Off' , S2:='$t', S3:= REAL_TO_STRING( EVP513.Cal_Off  ), S4:='$n', wSize := BUF_SIZE, pBuffer := ADR(aBuffer), wPos := wBufPos );
	F_ADD_STRINGX4_TO_BUFFER( S1:= 'EVP709_K'   , S2:='$t', S3:= REAL_TO_STRING( EVP709.Cal_K    ), S4:='$n', wSize := BUF_SIZE, pBuffer := ADR(aBuffer), wPos := wBufPos );
	F_ADD_STRINGX4_TO_BUFFER( S1:= 'EVP709_Off' , S2:='$t', S3:= REAL_TO_STRING( EVP709.Cal_Off  ), S4:='$n', wSize := BUF_SIZE, pBuffer := ADR(aBuffer), wPos := wBufPos );
	F_ADD_STRINGX4_TO_BUFFER( S1:= 'EVP1005_K'  , S2:='$t', S3:= REAL_TO_STRING( EVP1005.Cal_K   ), S4:='$n', wSize := BUF_SIZE, pBuffer := ADR(aBuffer), wPos := wBufPos );
	F_ADD_STRINGX4_TO_BUFFER( S1:= 'EVP1005_Off', S2:='$t', S3:= REAL_TO_STRING( EVP1005.Cal_Off ), S4:='$n', wSize := BUF_SIZE, pBuffer := ADR(aBuffer), wPos := wBufPos );
	F_ADD_STRINGX4_TO_BUFFER( S1:= 'EVP1010_K'  , S2:='$t', S3:= REAL_TO_STRING( EVP1010.Cal_K   ), S4:='$n', wSize := BUF_SIZE, pBuffer := ADR(aBuffer), wPos := wBufPos );
	F_ADD_STRINGX4_TO_BUFFER( S1:= 'EVP1010_Off', S2:='$t', S3:= REAL_TO_STRING( EVP1010.Cal_Off ), S4:='$n', wSize := BUF_SIZE, pBuffer := ADR(aBuffer), wPos := wBufPos );

	(*TANK + GS + MF00 + PP - Node36/37*)
	F_ADD_STRING_TO_BUFFER( S1:= '$n#TANK + GS + MF00 + PP - Node36/37:$n', wSize := BUF_SIZE, pBuffer := ADR(aBuffer), wPos := wBufPos );
	F_ADD_STRINGX4_TO_BUFFER( S1:= 'SF_Delay', S2:='$t', S3:= REAL_TO_STRING( SF_Delay ), S4:='$n', wSize := BUF_SIZE, pBuffer := ADR(aBuffer), wPos := wBufPos );

	F_WRITE_SENSOR_BAR ( BUF_SIZE, ADR(aBuffer), wBufPos, P010 );
	F_ADD_STRINGX4_TO_BUFFER( S1:= P010.Name , S2:='_Min$t', S3:= REAL_TO_STRING( P010.MinBar ), S4:='$n', wSize := BUF_SIZE, pBuffer := ADR(aBuffer), wPos := wBufPos );

	F_WRITE_SENSOR_TEMP( BUF_SIZE, ADR(aBuffer), wBufPos, S011 );
	F_WRITE_SENSOR_TEMP( BUF_SIZE, ADR(aBuffer), wBufPos, S100 );
	F_WRITE_SENSOR_TEMP( BUF_SIZE, ADR(aBuffer), wBufPos, S101 );
	F_WRITE_SENSOR_TEMP( BUF_SIZE, ADR(aBuffer), wBufPos, S102 );

	F_WRITE_SENSOR_BAR ( BUF_SIZE, ADR(aBuffer), wBufPos, P001 );
	F_WRITE_SENSOR_BAR ( BUF_SIZE, ADR(aBuffer), wBufPos, P002 );
	F_WRITE_SENSOR_BAR ( BUF_SIZE, ADR(aBuffer), wBufPos, P003 );
	F_WRITE_SENSOR_BAR ( BUF_SIZE, ADR(aBuffer), wBufPos, P051 );
	F_WRITE_SENSOR_BAR ( BUF_SIZE, ADR(aBuffer), wBufPos, P052 );

	(*Water Ballast*)
	F_ADD_STRING_TO_BUFFER( S1:= '$n#Water Ballast - Node30/32:$n', wSize := BUF_SIZE, pBuffer := ADR(aBuffer), wPos := wBufPos );
	F_WRITE_SENSOR_POS( BUF_SIZE, ADR(aBuffer), wBufPos, LS021 );
	F_WRITE_SENSOR_POS( BUF_SIZE, ADR(aBuffer), wBufPos, LS022 );
	F_WRITE_SENSOR_POS( BUF_SIZE, ADR(aBuffer), wBufPos, LS023 );
	F_WRITE_SENSOR_POS( BUF_SIZE, ADR(aBuffer), wBufPos, LS024 );

	(*MF01 - Node42*)
	F_ADD_STRING_TO_BUFFER( S1:= '$n#MF01 - Node42:$n', wSize := BUF_SIZE, pBuffer := ADR(aBuffer), wPos := wBufPos );
	F_WRITE_SENSOR_BAR( BUF_SIZE, ADR(aBuffer), wBufPos, P101 );
	F_WRITE_SENSOR_BAR( BUF_SIZE, ADR(aBuffer), wBufPos, P103 );

	(*MF02 - Node34*)
	F_ADD_STRING_TO_BUFFER( S1:= '$n#MF02 - Node34:$n', wSize := BUF_SIZE, pBuffer := ADR(aBuffer), wPos := wBufPos );
	F_WRITE_SENSOR_BAR( BUF_SIZE, ADR(aBuffer), wBufPos, P201  );

	(*MF03 - Node43/44*)
	F_ADD_STRING_TO_BUFFER( S1:= '$n#MF03 - Node43/44:$n', wSize := BUF_SIZE, pBuffer := ADR(aBuffer), wPos := wBufPos );
	F_WRITE_SENSOR_BAR( BUF_SIZE, ADR(aBuffer), wBufPos, P301 );
	F_WRITE_SENSOR_BAR( BUF_SIZE, ADR(aBuffer), wBufPos, P303 );
	F_WRITE_SENSOR_BAR( BUF_SIZE, ADR(aBuffer), wBufPos, P305 );
	F_WRITE_SENSOR_BAR( BUF_SIZE, ADR(aBuffer), wBufPos, P307 );
	F_WRITE_SENSOR_BAR( BUF_SIZE, ADR(aBuffer), wBufPos, P309 );
	F_WRITE_SENSOR_BAR( BUF_SIZE, ADR(aBuffer), wBufPos, P311 );

	F_WRITE_SENSOR_POS( BUF_SIZE, ADR(aBuffer), wBufPos, LS301 );
	F_WRITE_SENSOR_POS( BUF_SIZE, ADR(aBuffer), wBufPos, LS303 );
	F_WRITE_SENSOR_POS( BUF_SIZE, ADR(aBuffer), wBufPos, LS305 );
	F_WRITE_SENSOR_POS( BUF_SIZE, ADR(aBuffer), wBufPos, LS307 );
	F_WRITE_SENSOR_POS( BUF_SIZE, ADR(aBuffer), wBufPos, LS309 );
	F_WRITE_SENSOR_POS( BUF_SIZE, ADR(aBuffer), wBufPos, LS311 );

	F_WRITE_SENSOR_KG( BUF_SIZE, ADR(aBuffer), wBufPos, L301 );
	F_WRITE_SENSOR_KG( BUF_SIZE, ADR(aBuffer), wBufPos, L303 );
	F_WRITE_SENSOR_KG( BUF_SIZE, ADR(aBuffer), wBufPos, L305 );
	F_WRITE_SENSOR_KG( BUF_SIZE, ADR(aBuffer), wBufPos, L307 );
	F_WRITE_SENSOR_KG( BUF_SIZE, ADR(aBuffer), wBufPos, L309 );
	F_WRITE_SENSOR_KG( BUF_SIZE, ADR(aBuffer), wBufPos, L311 );

	(*MF05 - Node41*)
	F_ADD_STRING_TO_BUFFER( S1:= '$n#MF05 - Node41:$n', wSize := BUF_SIZE, pBuffer := ADR(aBuffer), wPos := wBufPos );
	F_WRITE_SENSOR_BAR( BUF_SIZE, ADR(aBuffer), wBufPos, P501 );
	F_WRITE_SENSOR_BAR( BUF_SIZE, ADR(aBuffer), wBufPos, P503 );
	F_WRITE_SENSOR_BAR( BUF_SIZE, ADR(aBuffer), wBufPos, P505 );
	F_WRITE_SENSOR_BAR( BUF_SIZE, ADR(aBuffer), wBufPos, P507 );

	F_WRITE_SENSOR_KG( BUF_SIZE, ADR(aBuffer), wBufPos, L501 );
	F_WRITE_SENSOR_KG( BUF_SIZE, ADR(aBuffer), wBufPos, L503 );
	F_WRITE_SENSOR_KG( BUF_SIZE, ADR(aBuffer), wBufPos, L505 );

	(*MF06 - Node20*)
	F_ADD_STRING_TO_BUFFER( S1:= '$n#MF06 - Node20:$n', wSize := BUF_SIZE, pBuffer := ADR(aBuffer), wPos := wBufPos );
	F_WRITE_SENSOR_BAR( BUF_SIZE, ADR(aBuffer), wBufPos, P601 );
	F_WRITE_SENSOR_BAR( BUF_SIZE, ADR(aBuffer), wBufPos, P603 );
	F_WRITE_SENSOR_BAR( BUF_SIZE, ADR(aBuffer), wBufPos, P605 );
	F_WRITE_SENSOR_BAR( BUF_SIZE, ADR(aBuffer), wBufPos, P607 );

	F_WRITE_SENSOR_POS( BUF_SIZE, ADR(aBuffer), wBufPos, LS601 );
	F_WRITE_SENSOR_POS( BUF_SIZE, ADR(aBuffer), wBufPos, LS605 );

	(*MF07 - Node21/22*)
	F_ADD_STRING_TO_BUFFER( S1:= '$n#MF07 - Node21/22:$n', wSize := BUF_SIZE, pBuffer := ADR(aBuffer), wPos := wBufPos );
	F_WRITE_SENSOR_BAR( BUF_SIZE, ADR(aBuffer), wBufPos, P701 );
	F_WRITE_SENSOR_BAR( BUF_SIZE, ADR(aBuffer), wBufPos, P703 );
	F_WRITE_SENSOR_BAR( BUF_SIZE, ADR(aBuffer), wBufPos, P705 );
	F_WRITE_SENSOR_BAR( BUF_SIZE, ADR(aBuffer), wBufPos, P707 );
	F_WRITE_SENSOR_BAR( BUF_SIZE, ADR(aBuffer), wBufPos, P709 );

	F_WRITE_SENSOR_POS( BUF_SIZE, ADR(aBuffer), wBufPos, LS707 );
	F_WRITE_SENSOR_POS( BUF_SIZE, ADR(aBuffer), wBufPos, LS709 );

	F_WRITE_SENSOR_KG( BUF_SIZE, ADR(aBuffer), wBufPos, L701 );
	F_WRITE_SENSOR_KG( BUF_SIZE, ADR(aBuffer), wBufPos, L703 );
	F_WRITE_SENSOR_KG( BUF_SIZE, ADR(aBuffer), wBufPos, L705 );
	F_WRITE_SENSOR_KG( BUF_SIZE, ADR(aBuffer), wBufPos, L707 );
	F_WRITE_SENSOR_KG( BUF_SIZE, ADR(aBuffer), wBufPos, L709 );

	(*MF08 - Node23*)
	F_ADD_STRING_TO_BUFFER( S1:= '$n#MF08 - Node23:$n', wSize := BUF_SIZE, pBuffer := ADR(aBuffer), wPos := wBufPos );
	F_WRITE_SENSOR_BAR( BUF_SIZE, ADR(aBuffer), wBufPos, P802 );
	F_WRITE_SENSOR_BAR( BUF_SIZE, ADR(aBuffer), wBufPos, P804 );

	F_WRITE_SENSOR_POS( BUF_SIZE, ADR(aBuffer), wBufPos, LS801 );
	F_WRITE_SENSOR_POS( BUF_SIZE, ADR(aBuffer), wBufPos, LS803 );

	F_WRITE_SENSOR_KG( BUF_SIZE, ADR(aBuffer), wBufPos, L901 );
	F_WRITE_SENSOR_KG( BUF_SIZE, ADR(aBuffer), wBufPos, L903 );

	(*MF09 - Node35*)
	F_ADD_STRING_TO_BUFFER( S1:= '$n#MF09 - Node35:$n', wSize := BUF_SIZE, pBuffer := ADR(aBuffer), wPos := wBufPos );
	F_WRITE_SENSOR_BAR( BUF_SIZE, ADR(aBuffer), wBufPos, P901 );
	F_WRITE_SENSOR_BAR( BUF_SIZE, ADR(aBuffer), wBufPos, P903 );

	F_WRITE_SENSOR_POS( BUF_SIZE, ADR(aBuffer), wBufPos, LS901 );
	F_WRITE_SENSOR_POS( BUF_SIZE, ADR(aBuffer), wBufPos, LS903 );

	(*MF10 - Node40*)
	F_ADD_STRING_TO_BUFFER( S1:= '$n#MF10 - Node40:$n', wSize := BUF_SIZE, pBuffer := ADR(aBuffer), wPos := wBufPos );
	F_WRITE_SENSOR_BAR( BUF_SIZE, ADR(aBuffer), wBufPos, P1001 );
	F_WRITE_SENSOR_BAR( BUF_SIZE, ADR(aBuffer), wBufPos, P1002 );

	F_WRITE_SENSOR_POS( BUF_SIZE, ADR(aBuffer), wBufPos, LS1001 );
	F_WRITE_SENSOR_POS( BUF_SIZE, ADR(aBuffer), wBufPos, LS1002 );

	(*MF11 - Node21*)
	F_ADD_STRING_TO_BUFFER( S1:= '$n#MF11 - Node21:$n', wSize := BUF_SIZE, pBuffer := ADR(aBuffer), wPos := wBufPos );
	F_WRITE_SENSOR_BAR ( BUF_SIZE, ADR(aBuffer), wBufPos, P1101 );
	F_WRITE_SENSOR_BAR ( BUF_SIZE, ADR(aBuffer), wBufPos, P1102 );
	F_WRITE_SENSOR_TEMP( BUF_SIZE, ADR(aBuffer), wBufPos, S1100 );


	(*MF12 - Node24/25*)
	F_ADD_STRING_TO_BUFFER( S1:= '$n#MF12 - Node24/25:$n', wSize := BUF_SIZE, pBuffer := ADR(aBuffer), wPos := wBufPos );
	F_WRITE_SENSOR_BAR( BUF_SIZE, ADR(aBuffer), wBufPos, P1202 );
	F_WRITE_SENSOR_BAR( BUF_SIZE, ADR(aBuffer), wBufPos, P1203 );
	F_WRITE_SENSOR_BAR( BUF_SIZE, ADR(aBuffer), wBufPos, P1204 );
	F_WRITE_SENSOR_BAR( BUF_SIZE, ADR(aBuffer), wBufPos, P1205 );
	F_WRITE_SENSOR_BAR( BUF_SIZE, ADR(aBuffer), wBufPos, P1206 );
	F_WRITE_SENSOR_BAR( BUF_SIZE, ADR(aBuffer), wBufPos, P1207 );
	F_WRITE_SENSOR_BAR( BUF_SIZE, ADR(aBuffer), wBufPos, P1208 );
	F_WRITE_SENSOR_BAR( BUF_SIZE, ADR(aBuffer), wBufPos, P1209 );
	F_WRITE_SENSOR_BAR( BUF_SIZE, ADR(aBuffer), wBufPos, P1210 );
	F_WRITE_SENSOR_BAR( BUF_SIZE, ADR(aBuffer), wBufPos, P1211 );
	F_WRITE_SENSOR_BAR( BUF_SIZE, ADR(aBuffer), wBufPos, P1212 );
	F_WRITE_SENSOR_BAR( BUF_SIZE, ADR(aBuffer), wBufPos, P1213 );
	F_WRITE_SENSOR_BAR( BUF_SIZE, ADR(aBuffer), wBufPos, P1214 );
	F_WRITE_SENSOR_BAR( BUF_SIZE, ADR(aBuffer), wBufPos, P1215 );
	F_WRITE_SENSOR_BAR( BUF_SIZE, ADR(aBuffer), wBufPos, P1216 );
	F_WRITE_SENSOR_BAR( BUF_SIZE, ADR(aBuffer), wBufPos, P1219 );

	(*MF13 - Node33 - Traveller*)
	F_ADD_STRING_TO_BUFFER( S1:= '$n#MF13 - Node33:$n', wSize := BUF_SIZE, pBuffer := ADR(aBuffer), wPos := wBufPos );
	F_WRITE_SENSOR_BAR( BUF_SIZE, ADR(aBuffer), wBufPos, P1301 );
	F_WRITE_SENSOR_BAR( BUF_SIZE, ADR(aBuffer), wBufPos, P1302 );

	F_WRITE_SENSOR_POS( BUF_SIZE, ADR(aBuffer), wBufPos, LS1303 );

	(*MF16 - Node34*)
	F_ADD_STRING_TO_BUFFER( S1:= '$n#MF16 - Node34:$n', wSize := BUF_SIZE, pBuffer := ADR(aBuffer), wPos := wBufPos );
	F_WRITE_SENSOR_BAR( BUF_SIZE, ADR(aBuffer), wBufPos, P1602 );
	F_WRITE_SENSOR_BAR( BUF_SIZE, ADR(aBuffer), wBufPos, P1603 );
	F_WRITE_SENSOR_BAR( BUF_SIZE, ADR(aBuffer), wBufPos, P1604 );
	F_WRITE_SENSOR_BAR( BUF_SIZE, ADR(aBuffer), wBufPos, P1605 );

	(*MF19 - Node32*)
	F_ADD_STRING_TO_BUFFER( S1:= '$n#MF19 - Node32:$n', wSize := BUF_SIZE, pBuffer := ADR(aBuffer), wPos := wBufPos );
	F_WRITE_SENSOR_POS( BUF_SIZE, ADR(aBuffer), wBufPos, LS1905 );

	(*MF20 - Node31*)
	F_ADD_STRING_TO_BUFFER( S1:= '$n#MF20 - Node31:$n', wSize := BUF_SIZE, pBuffer := ADR(aBuffer), wPos := wBufPos );
	F_WRITE_SENSOR_POS( BUF_SIZE, ADR(aBuffer), wBufPos, LS2001 );
	F_WRITE_SENSOR_POS( BUF_SIZE, ADR(aBuffer), wBufPos, LS2005 );

	(*MF22 - Node29*)
	F_ADD_STRING_TO_BUFFER( S1:= '$n#MF22 - Node29:$n', wSize := BUF_SIZE, pBuffer := ADR(aBuffer), wPos := wBufPos );
	F_WRITE_SENSOR_POS( BUF_SIZE, ADR(aBuffer), wBufPos, LS2201 );

	(*MF23 - Node30*)
	F_ADD_STRING_TO_BUFFER( S1:= '$n#MF23 - Node30:$n', wSize := BUF_SIZE, pBuffer := ADR(aBuffer), wPos := wBufPos );
	F_WRITE_SENSOR_POS( BUF_SIZE, ADR(aBuffer), wBufPos, LS2301 );
	F_WRITE_SENSOR_POS( BUF_SIZE, ADR(aBuffer), wBufPos, LS2305 );

	(*MF24 - Node29*)
	F_ADD_STRING_TO_BUFFER( S1:= '$n#MF24 - Node29:$n', wSize := BUF_SIZE, pBuffer := ADR(aBuffer), wPos := wBufPos );
	F_WRITE_SENSOR_POS( BUF_SIZE, ADR(aBuffer), wBufPos, LS2401 );
	F_WRITE_SENSOR_POS( BUF_SIZE, ADR(aBuffer), wBufPos, LS2409 );

	(*MF25 - Node26*)
	F_ADD_STRING_TO_BUFFER( S1:= '$n#MF25 - Node26:$n', wSize := BUF_SIZE, pBuffer := ADR(aBuffer), wPos := wBufPos );
	F_WRITE_SENSOR_BAR( BUF_SIZE, ADR(aBuffer), wBufPos,  P2500 );
	F_WRITE_SENSOR_POS( BUF_SIZE, ADR(aBuffer), wBufPos, LS2501 );
	F_WRITE_SENSOR_POS( BUF_SIZE, ADR(aBuffer), wBufPos, LS2505 );

	(*DGB Seal - Node48*)
	F_WRITE_SENSOR_BAR ( BUF_SIZE, ADR(aBuffer), wBufPos, P_SealP );
	F_WRITE_SENSOR_BAR ( BUF_SIZE, ADR(aBuffer), wBufPos, P_SealS );


	(*Next State*)
	State := 210;

210: (*Save Sensors Buffer*)
	fbSaveList( bEnable:= TRUE, pBuffer:= ADR(aBuffer), wBufLen:= wBufPos );

	IF fbSaveList.bDone THEN
		State  := 220;
	END_IF

220: (*Create Parameters Buffer*)
	fbSaveList( bEnable:= FALSE );
	fbSaveList.sFilePath := '\Hard Disk\FTP\';
	fbSaveList.sFileName := 'Parameters';
	fbSaveList.sFileExt  := '.txt';
	fbSaveList.Backup    := TRUE;

	wBufPos := 0;

(*1-Engine*)
	F_WRITE_ENGINE_CFG    ( 'Engine'    , BUF_SIZE, ADR(aBuffer), wBufPos, stEngineCfg     );
	F_WRITE_POWERPACK_CFG ( 'Powerpack' , BUF_SIZE, ADR(aBuffer), wBufPos, stPowerpackCfg  );
	F_WRITE_PROPULSION_CFG( 'Propulsion', BUF_SIZE, ADR(aBuffer), wBufPos, stPropulsionCfg );

(*2- HP Fucntions*)
	F_WRITE_SE_CYLINDER_POS_CFG	( 'A3Tack', BUF_SIZE, ADR(aBuffer), wBufPos, stSE301Cfg   );
	F_WRITE_SE_CYLINDER_POS_CFG	( 'FrTack', BUF_SIZE, ADR(aBuffer), wBufPos, stSE303Cfg   );
	F_WRITE_SE_CYLINDER_POS_CFG	( 'J5'    , BUF_SIZE, ADR(aBuffer), wBufPos, stSE305Cfg   );
	F_WRITE_SE_CYLINDER_POS_CFG	( 'J4'    , BUF_SIZE, ADR(aBuffer), wBufPos, stSE307Cfg   );
	F_WRITE_SE_CYLINDER_POS_CFG ( 'Fsy'   , BUF_SIZE, ADR(aBuffer), wBufPos, stSE309Cfg   );
	F_WRITE_SE_CYLINDER_POS_CFG	( 'J2'    , BUF_SIZE, ADR(aBuffer), wBufPos, stSE311Cfg   );

	F_WRITE_SE_CYLINDER_CFG		( 'JibIO' , BUF_SIZE, ADR(aBuffer), wBufPos, stSE501Cfg   );
	F_WRITE_SE_CYLINDER_CFG		( 'JibUD' , BUF_SIZE, ADR(aBuffer), wBufPos, stSE503Cfg   );
	F_WRITE_SE_CYLINDER_CFG		( 'Vang'  , BUF_SIZE, ADR(aBuffer), wBufPos, stSE505Cfg   );

	F_WRITE_LIFT_PROP_CFG       ( 'PropUpDw', BUF_SIZE, ADR(aBuffer), wBufPos, stDE601Cfg );
	F_WRITE_DE_CYLINDER_POS_CFG	( 'TrimTab' , BUF_SIZE, ADR(aBuffer), wBufPos, stDE605Cfg );

	F_WRITE_SE_CYLINDER_CFG		( 'Inn'   , BUF_SIZE, ADR(aBuffer), wBufPos, stSE701Cfg   );
	F_WRITE_SE_CYLINDER_CFG		( 'Out'   , BUF_SIZE, ADR(aBuffer), wBufPos, stSE703Cfg   );
	F_WRITE_SE_CYLINDER_CFG		( 'Cunn'  , BUF_SIZE, ADR(aBuffer), wBufPos, stSE705Cfg   );
	F_WRITE_SE_CYLINDER_POS_CFG	( 'Runn'  , BUF_SIZE, ADR(aBuffer), wBufPos, stSE707Cfg   );
	F_WRITE_SE_CYLINDER_POS_CFG	( 'Chksy' , BUF_SIZE, ADR(aBuffer), wBufPos, stSE709Cfg   );

	F_WRITE_SE_CYLINDER_POS_CFG	( 'BsyP'  , BUF_SIZE, ADR(aBuffer), wBufPos, stSE901Cfg   );
	(*F_WRITE_SE_CYLINDER_POS_CFG	( 'BsyS'  , BUF_SIZE, ADR(aBuffer), wBufPos, stSE903Cfg   );*)

(*3- Water Ballast*)
	F_WRITE_WB_CFG        ( 'WB'        , BUF_SIZE, ADR(aBuffer), wBufPos, stWBCfg        );
	F_WRITE_WB_VALVESF_CFG( 'WBValves'  , BUF_SIZE, ADR(aBuffer), wBufPos, stWBValveSFCfg );
	F_WRITE_WB_VALVELS_CFG( 'WBValvesLS', BUF_SIZE, ADR(aBuffer), wBufPos, stWBValveLSCfg );

(*4- LP Functions*)
	F_WRITE_WINCHE_CFG ( 'W1202', BUF_SIZE, ADR(aBuffer), wBufPos, stW1202Cfg );
	F_WRITE_WINCHE_CFG ( 'W1204', BUF_SIZE, ADR(aBuffer), wBufPos, stW1204Cfg );
	F_WRITE_WINCHE_CFG ( 'W1206', BUF_SIZE, ADR(aBuffer), wBufPos, stW1206Cfg );
	F_WRITE_WINCHE_CFG ( 'W1208', BUF_SIZE, ADR(aBuffer), wBufPos, stW1208Cfg );
	F_WRITE_WINCHE_CFG ( 'W1210', BUF_SIZE, ADR(aBuffer), wBufPos, stW1210Cfg );
	F_WRITE_WINCHE_CFG ( 'W1212', BUF_SIZE, ADR(aBuffer), wBufPos, stW1212Cfg );
	F_WRITE_WINCHE_CFG ( 'W1214', BUF_SIZE, ADR(aBuffer), wBufPos, stW1214Cfg );
	F_WRITE_WINCHE_CFG ( 'W1602', BUF_SIZE, ADR(aBuffer), wBufPos, stW1602Cfg );
	F_WRITE_WINCHE_CFG ( 'W1604', BUF_SIZE, ADR(aBuffer), wBufPos, stW1604Cfg );

	F_ADD_STRINGX4_TO_BUFFER( S1:= 'WRAMP_Min', S2:='$t', S3:= REAL_TO_STRING( stWRampCfg.Spd_Min), S4:='$n', wSize := BUF_SIZE, pBuffer := ADR(aBuffer), wPos := wBufPos );
	F_ADD_STRINGX4_TO_BUFFER( S1:= 'WRAMP_Inc', S2:='$t', S3:= REAL_TO_STRING( stWRampCfg.Spd_Inc), S4:='$n', wSize := BUF_SIZE, pBuffer := ADR(aBuffer), wPos := wBufPos );
	F_ADD_STRINGX4_TO_BUFFER( S1:= 'WRAMP_Dec', S2:='$t', S3:= REAL_TO_STRING( stWRampCfg.Spd_Dec), S4:='$n', wSize := BUF_SIZE, pBuffer := ADR(aBuffer), wPos := wBufPos );

	F_WRITE_BOARD_CFG     ( 'Board'    , BUF_SIZE, ADR(aBuffer), wBufPos, stBoardCfg     );
	F_WRITE_KEEL_CFG      ( 'Keel'     , BUF_SIZE, ADR(aBuffer), wBufPos, stKeelCfg      );
	F_WRITE_TRAVELLER_CFG ( 'Traveller', BUF_SIZE, ADR(aBuffer), wBufPos, stTravellerCfg );

	F_WRITE_LP_FUNC_CFG ( 'BowThr'    , BUF_SIZE, ADR(aBuffer), wBufPos, stBowThrCfg     );
	F_WRITE_LP_FUNC_CFG ( 'BowThrUpDw', BUF_SIZE, ADR(aBuffer), wBufPos, stBowThrUpDwCfg );

	F_WRITE_TACK_VALVE_CFG ( 'TackValve', BUF_SIZE, ADR(aBuffer), wBufPos, stTackValveCfg );

	F_WRITE_MAST_SETUP_CFG ( 'MastSetup', BUF_SIZE, ADR(aBuffer), wBufPos, stMastSetup );


(*UDP Parameters*)
	F_ADD_STRING_TO_BUFFER  ( S1:= '$n#UDP Parameters:$n', wSize := BUF_SIZE, pBuffer := ADR(aBuffer), wPos := wBufPos );

	F_ADD_STRINGX4_TO_BUFFER( S1:= 'UDPHost', S2:='$t', S3:= sUDPSendHost                   , S4:='$n', wSize := BUF_SIZE, pBuffer := ADR(aBuffer), wPos := wBufPos );
	F_ADD_STRINGX4_TO_BUFFER( S1:= 'UDPPort', S2:='$t', S3:= UDINT_TO_STRING( nUDPSendPort ), S4:='$n', wSize := BUF_SIZE, pBuffer := ADR(aBuffer), wPos := wBufPos );
	F_ADD_STRINGX4_TO_BUFFER( S1:= 'UDPTime', S2:='$t', S3:= UINT_TO_STRING ( nUDPSendTime ), S4:='$n$n', wSize := BUF_SIZE, pBuffer := ADR(aBuffer), wPos := wBufPos );
	F_ADD_STRINGX4_TO_BUFFER( S1:= 'UDPRecvPort', S2:='$t', S3:= UDINT_TO_STRING( nUDPRecvPort ), S4:='$n', wSize := BUF_SIZE, pBuffer := ADR(aBuffer), wPos := wBufPos );

	F_ADD_STRINGX4_TO_BUFFER( S1:= 'UDPAlarmsHost', S2:='$t', S3:= sUDPAlarmsHost                   , S4:='$n', wSize := BUF_SIZE, pBuffer := ADR(aBuffer), wPos := wBufPos );
	F_ADD_STRINGX4_TO_BUFFER( S1:= 'UDPAlarmsPort', S2:='$t', S3:= UDINT_TO_STRING( nUDPAlarmsPort ), S4:='$n', wSize := BUF_SIZE, pBuffer := ADR(aBuffer), wPos := wBufPos );

	(*Next State*)
	State := 230;


230: (*Save PArameters Buffer*)
	fbSaveList( bEnable:= TRUE, pBuffer:= ADR(aBuffer), wBufLen:= wBufPos );

	IF fbSaveList.bDone THEN
		(*Loaded := FALSE;*)	(*No hace falta hacer el Reload despues de save.*)
								(*En CK las rampas las calulo siempre.*)
		State  := 300;
	END_IF


300: (*Calule coefficents*)
	F_CALC_ENGINE_COEF    ( Cycle:= MAIN.Cycle_Time, Cfg:= stEngineCfg     );
	F_CALC_PROPULSION_COEF(                          Cfg:= stPropulsionCfg );
	F_CALC_KEEL_COEF      (                          Cfg:= stKeelCfg       );

	(*Next State*)
	Loaded := TRUE;
	State  := 0;

END_CASE
END_PROGRAM

(* POU FUN/PARAMETERS/F_READ_SENSOR_BAR, ST *)
FUNCTION F_READ_SENSOR_BAR : BOOL
VAR_INPUT
END_VAR
VAR_IN_OUT
	stSensor : ST_SENSOR_BAR;
	fbIdList : FB_IDLIST;
END_VAR
VAR
END_VAR
stSensor.Cal_K   := F_IDLIST_GETREAL( CONCAT(stSensor.Name, '_K'   ), fbIdList );
stSensor.Cal_Off := stSensor.Cal_K * -stSensor.Raw_Off;
stSensor.MaxBar  := F_IDLIST_GETREAL( CONCAT(stSensor.Name, '_Max' ), fbIdList );
END_FUNCTION

(* POU FUN/PARAMETERS/F_READ_SENSOR_TEMP, ST *)
FUNCTION F_READ_SENSOR_TEMP : BOOL
VAR_INPUT
END_VAR
VAR_IN_OUT
	stSensor : ST_SENSOR_TEMP;
	fbIdList : FB_IDLIST;
END_VAR
VAR
END_VAR
stSensor.Cal_K   := F_IDLIST_GETREAL( CONCAT(stSensor.Name, '_K'   ), fbIdList );
stSensor.Cal_Off := F_IDLIST_GETREAL( CONCAT(stSensor.Name, '_Off' ), fbIdList );

stSensor.LowDeg  := F_IDLIST_GETREAL( CONCAT(stSensor.Name, '_Mild' ), fbIdList );
stSensor.HigDeg  := F_IDLIST_GETREAL( CONCAT(stSensor.Name, '_High' ), fbIdList );
stSensor.MaxDeg  := F_IDLIST_GETREAL( CONCAT(stSensor.Name, '_Max'  ), fbIdList );
stSensor.Delay   := F_IDLIST_GETREAL( CONCAT(stSensor.Name, '_Dly'  ), fbIdList );
END_FUNCTION

(* POU FUN/PARAMETERS/F_READ_SENSOR_POS, ST *)
FUNCTION F_READ_SENSOR_POS : BOOL
VAR_INPUT
END_VAR
VAR_IN_OUT
	stSensor : ST_SENSOR_POS;
	fbIdList : FB_IDLIST;
END_VAR
VAR
END_VAR
stSensor.Cal_K   := F_IDLIST_GETREAL( CONCAT(stSensor.Name, '_K'   ), fbIdList );
stSensor.Cal_Off := F_IDLIST_GETREAL( CONCAT(stSensor.Name, '_Off' ), fbIdList );
END_FUNCTION

(* POU FUN/PARAMETERS/F_READ_SENSOR_KG, ST *)
FUNCTION F_READ_SENSOR_KG : BOOL
VAR_INPUT
END_VAR
VAR_IN_OUT
	stSensor : ST_SENSOR_KG;
	fbIdList : FB_IDLIST;
END_VAR
VAR
END_VAR
stSensor.Cal_K := F_IDLIST_GETREAL( CONCAT(stSensor.Name, '_K' ), fbIdList );
stSensor.Cal_C := F_IDLIST_GETREAL( CONCAT(stSensor.Name, '_C' ), fbIdList );
END_FUNCTION

(* POU FUN/PARAMETERS/F_READ_ENGINE_CFG, ST *)
FUNCTION F_READ_ENGINE_CFG : BOOL
VAR_INPUT
	sHead : STRING;
	rTime : REAL;
END_VAR
VAR_IN_OUT
	stEngineCfg : ST_ENGINE_CFG;
	fbParamList : FB_IDLIST;
END_VAR
VAR
END_VAR
stEngineCfg.Min_RPM    := F_IDLIST_GETREAL( CONCAT(sHead, '_Min_RPM'   ), fbParamList );
stEngineCfg.Max_RPM    := F_IDLIST_GETREAL( CONCAT(sHead, '_Max_RPM'   ), fbParamList );
stEngineCfg.Boost_RPM  := F_IDLIST_GETREAL( CONCAT(sHead, '_Boost_RPM' ), fbParamList );
stEngineCfg.Stop_RPM   := F_IDLIST_GETREAL( CONCAT(sHead, '_Stop_RPM'  ), fbParamList );
stEngineCfg.MaxInc_RPM := F_IDLIST_GETREAL( CONCAT(sHead, '_MaxInc_RPM'), fbParamList );
stEngineCfg.MaxDec_RPM := F_IDLIST_GETREAL( CONCAT(sHead, '_MaxDec_RPM'), fbParamList );
stEngineCfg.DlyDec_sec := F_IDLIST_GETREAL( CONCAT(sHead, '_DlyDec_sec'), fbParamList );

stEngineCfg.HP_Nx_RPM := F_IDLIST_GETREAL( CONCAT(sHead, '_HP_Nx_RPM'), fbParamList );
stEngineCfg.HP_SF_RPM := F_IDLIST_GETREAL( CONCAT(sHead, '_HP_SF_RPM'), fbParamList );

stEngineCfg.LP_CK_RPM := F_IDLIST_GETREAL( CONCAT(sHead, '_LP_CK_RPM'), fbParamList );
stEngineCfg.LP_1x_RPM := F_IDLIST_GETREAL( CONCAT(sHead, '_LP_1x_RPM'), fbParamList );
stEngineCfg.LP_2x_RPM := F_IDLIST_GETREAL( CONCAT(sHead, '_LP_2x_RPM'), fbParamList );
stEngineCfg.LP_3x_RPM := F_IDLIST_GETREAL( CONCAT(sHead, '_LP_3x_RPM'), fbParamList );
stEngineCfg.LP_Nx_RPM := F_IDLIST_GETREAL( CONCAT(sHead, '_LP_Nx_RPM'), fbParamList );

stEngineCfg.N_Winch_WOP := F_IDLIST_GETINT( CONCAT(sHead, '_N_WinchWOP'), fbParamList );
stEngineCfg.N_Winch_WK  := F_IDLIST_GETINT( CONCAT(sHead, '_N_WinchWK' ), fbParamList );
stEngineCfg.N_Winch_WP  := F_IDLIST_GETINT( CONCAT(sHead, '_N_WinchWP' ), fbParamList );

stEngineCfg.Max_Torque := F_IDLIST_GETREAL( CONCAT(sHead, '_Max_Torque'), fbParamList );
stEngineCfg.Min_Torque := F_IDLIST_GETREAL( CONCAT(sHead, '_Min_Torque'), fbParamList );

stEngineCfg.Inc_RMP_Perc_WOP := F_IDLIST_GETREAL( CONCAT(sHead, '_Inc_RMP_Perc_WOP'), fbParamList );
stEngineCfg.Dec_Flow_Perc_WP := F_IDLIST_GETREAL( CONCAT(sHead, '_Dec_Flow_Perc_WP'), fbParamList );

stEngineCfg.Max_HeatExch_P := F_IDLIST_GETREAL( CONCAT(sHead, '_Max_HeatExch_P' ), fbParamList );

stEngineCfg.EnForceRPM := F_IDLIST_GETBOOL( CONCAT(sHead, '_EnForceRPM' ), fbParamList );
stEngineCfg.EnForceTHR := F_IDLIST_GETBOOL( CONCAT(sHead, '_EnForceTHR' ), fbParamList );

stEngineCfg.Cycle := rTime;
END_FUNCTION

(* POU FUN/PARAMETERS/F_READ_POWERPACK_CFG, ST *)
FUNCTION F_READ_POWERPACK_CFG : BOOL
VAR_INPUT
	sHead : STRING;
	rTime : REAL;
END_VAR
VAR_IN_OUT
	stConfig : ST_POWERPACK_CFG;
	fbIdList : FB_IDLIST;
END_VAR
VAR
END_VAR
stConfig.Hyst_HP := F_IDLIST_GETREAL( CONCAT(sHead, '_Hyst_HP' ), fbIdList );
stConfig.Hyst_LP := F_IDLIST_GETREAL( CONCAT(sHead, '_Hyst_LP' ), fbIdList );
stConfig.Hyst_TM := F_IDLIST_GETREAL( CONCAT(sHead, '_Hyst_TM' ), fbIdList );
stConfig.Thr_HP  := F_IDLIST_GETREAL( CONCAT(sHead, '_Thr_HP'  ), fbIdList );
stConfig.Thr_LP  := F_IDLIST_GETREAL( CONCAT(sHead, '_Thr_LP'  ), fbIdList );
stConfig.Cycle   := rTime;
END_FUNCTION

(* POU FUN/PARAMETERS/F_READ_PROPULSION_CFG, ST *)
FUNCTION F_READ_PROPULSION_CFG : BOOL
VAR_INPUT
	sHead : STRING;
	rTime : REAL;
END_VAR
VAR_IN_OUT
	stPropulsionCfg : ST_PROPULSION_CFG;
	fbParamList     : FB_IDLIST;
END_VAR
VAR
END_VAR
stPropulsionCfg.aThrt_V[0]  := F_IDLIST_GETREAL( CONCAT(sHead, '_Thrt0_V' ), fbParamList );
stPropulsionCfg.aThrt_V[4]  := F_IDLIST_GETREAL( CONCAT(sHead, '_Thrt4_V' ), fbParamList );
stPropulsionCfg.aThrt_V[5]  := F_IDLIST_GETREAL( CONCAT(sHead, '_Thrt5_V' ), fbParamList );
stPropulsionCfg.aThrt_V[6]  := F_IDLIST_GETREAL( CONCAT(sHead, '_Thrt6_V' ), fbParamList );
stPropulsionCfg.aThrt_V[10] := F_IDLIST_GETREAL( CONCAT(sHead, '_Thrt10_V'), fbParamList );
stPropulsionCfg.IdleDB_V    := F_IDLIST_GETREAL( CONCAT(sHead, '_ThrDB_V' ), fbParamList );

stPropulsionCfg.PropRPM_K   := F_IDLIST_GETREAL( CONCAT(sHead, '_RPM_K' ), fbParamList );
stPropulsionCfg.Delay_Off   := F_IDLIST_GETREAL( CONCAT(sHead, '_Delay_Off' ), fbParamList );
stPropulsionCfg.Cycle       := rTime;

stPropulsionCfg.aEng_RPM[0]  := F_IDLIST_GETREAL( CONCAT(sHead, '_RPM0' ), fbParamList );
stPropulsionCfg.aEng_RPM[1]  := F_IDLIST_GETREAL( CONCAT(sHead, '_RPM1' ), fbParamList );
stPropulsionCfg.aEng_RPM[2]  := F_IDLIST_GETREAL( CONCAT(sHead, '_RPM2' ), fbParamList );
stPropulsionCfg.aEng_RPM[3]  := F_IDLIST_GETREAL( CONCAT(sHead, '_RPM3' ), fbParamList );
stPropulsionCfg.aEng_RPM[4]  := F_IDLIST_GETREAL( CONCAT(sHead, '_RPM4' ), fbParamList );
stPropulsionCfg.aEng_RPM[5]  := 0.0;
stPropulsionCfg.aEng_RPM[6]  := F_IDLIST_GETREAL( CONCAT(sHead, '_RPM6' ), fbParamList );
stPropulsionCfg.aEng_RPM[7]  := F_IDLIST_GETREAL( CONCAT(sHead, '_RPM7' ), fbParamList );
stPropulsionCfg.aEng_RPM[8]  := F_IDLIST_GETREAL( CONCAT(sHead, '_RPM8' ), fbParamList );
stPropulsionCfg.aEng_RPM[9]  := F_IDLIST_GETREAL( CONCAT(sHead, '_RPM9' ), fbParamList );
stPropulsionCfg.aEng_RPM[10] := F_IDLIST_GETREAL( CONCAT(sHead, '_RPM10'), fbParamList );

stPropulsionCfg.aEVP_mA[0]  := F_IDLIST_GETREAL( CONCAT(sHead, '_EVP0_mA' ), fbParamList );
stPropulsionCfg.aEVP_mA[1]  := F_IDLIST_GETREAL( CONCAT(sHead, '_EVP1_mA' ), fbParamList );
stPropulsionCfg.aEVP_mA[2]  := F_IDLIST_GETREAL( CONCAT(sHead, '_EVP2_mA' ), fbParamList );
stPropulsionCfg.aEVP_mA[3]  := F_IDLIST_GETREAL( CONCAT(sHead, '_EVP3_mA' ), fbParamList );
stPropulsionCfg.aEVP_mA[4]  := F_IDLIST_GETREAL( CONCAT(sHead, '_EVP4_mA' ), fbParamList );
stPropulsionCfg.aEVP_mA[5]  := 0.0;
stPropulsionCfg.aEVP_mA[6]  := F_IDLIST_GETREAL( CONCAT(sHead, '_EVP6_mA' ), fbParamList );
stPropulsionCfg.aEVP_mA[7]  := F_IDLIST_GETREAL( CONCAT(sHead, '_EVP7_mA' ), fbParamList );
stPropulsionCfg.aEVP_mA[8]  := F_IDLIST_GETREAL( CONCAT(sHead, '_EVP8_mA' ), fbParamList );
stPropulsionCfg.aEVP_mA[9]  := F_IDLIST_GETREAL( CONCAT(sHead, '_EVP9_mA' ), fbParamList );
stPropulsionCfg.aEVP_mA[10] := F_IDLIST_GETREAL( CONCAT(sHead, '_EVP10_mA'), fbParamList );
END_FUNCTION

(* POU FUN/PARAMETERS/F_READ_SE_CYLINDER_POS_CFG, ST *)
FUNCTION F_READ_SE_CYLINDER_POS_CFG : BOOL
VAR_INPUT
	sHead : STRING;
	rTime : REAL;
END_VAR
VAR_IN_OUT
	stConfig : ST_SE_CYLINDER_POS_CFG;
	fbIdList : FB_IDLIST;
END_VAR
VAR
	SMax: BOOL;
END_VAR
stConfig.Ease    := F_IDLIST_GETREAL( CONCAT(sHead, '_Ease'    ), fbIdList );

stConfig.TgtLS_In  := F_IDLIST_GETREAL( CONCAT(sHead, '_TgtLS_In'  ), fbIdList );
stConfig.TgtLS_Out := F_IDLIST_GETREAL( CONCAT(sHead, '_TgtLS_Out' ), fbIdList );
stConfig.TgtLS_Slow := F_IDLIST_GETREAL( CONCAT(sHead, '_TgtLS_Slow' ), fbIdList );

stConfig.TimeMax  := F_IDLIST_GETREAL( CONCAT(sHead, '_TimeMax'  ), fbIdList );
stConfig.TimeEase := F_IDLIST_GETREAL( CONCAT(sHead, '_TimeEase' ), fbIdList );
stConfig.Cycle    := rTime;

stConfig.LS_Limit_In  := F_IDLIST_GETBOOL( CONCAT(sHead, '_LS_Limit_In'  ), fbIdList );
stConfig.LS_Limit_Out := F_IDLIST_GETBOOL( CONCAT(sHead, '_LS_Limit_Out' ), fbIdList );

stConfig.HP  := F_IDLIST_GETBYTE( CONCAT(sHead, '_HP'  ), fbIdList );
END_FUNCTION

(* POU FUN/PARAMETERS/F_READ_SE_CYLINDER_CFG, ST *)
FUNCTION F_READ_SE_CYLINDER_CFG : BOOL
VAR_INPUT
	sHead : STRING;
	rTime : REAL;
END_VAR
VAR_IN_OUT
	stConfig : ST_SE_CYLINDER_CFG;
	fbIdList : FB_IDLIST;
END_VAR
stConfig.Ease     := F_IDLIST_GETREAL( CONCAT(sHead, '_Ease'     ), fbIdList );
stConfig.TimeMax  := F_IDLIST_GETREAL( CONCAT(sHead, '_TimeMax'  ), fbIdList );
stConfig.TimeEase := F_IDLIST_GETREAL( CONCAT(sHead, '_TimeEase' ), fbIdList );
stConfig.HP       := F_IDLIST_GETBYTE( CONCAT(sHead, '_HP'       ), fbIdList );
stConfig.Cycle    := rTime;
END_FUNCTION

(* POU FUN/PARAMETERS/F_READ_LIFT_PROP_CFG, ST *)
FUNCTION F_READ_LIFT_PROP_CFG : BOOL
VAR_INPUT
	sHead : STRING;
	rTime : REAL;
END_VAR
VAR_IN_OUT
	stConfig : ST_LIFT_PROP_CFG;
	fbIdList : FB_IDLIST;
END_VAR
VAR
END_VAR
stConfig.TgtP_Up  := F_IDLIST_GETREAL( CONCAT(sHead, '_TgtP_Up'  ), fbIdList );
stConfig.TgtP_Dw  := F_IDLIST_GETREAL( CONCAT(sHead, '_TgtP_Dw'  ), fbIdList );
stConfig.TgtLS_Up := F_IDLIST_GETREAL( CONCAT(sHead, '_TgtLS_Up' ), fbIdList );
stConfig.TgtLS_Dw := F_IDLIST_GETREAL( CONCAT(sHead, '_TgtLS_Dw' ), fbIdList );

stConfig.P_DB     := F_IDLIST_GETREAL( CONCAT(sHead, '_P_DB'     ), fbIdList );
stConfig.LS_DB    := F_IDLIST_GETREAL( CONCAT(sHead, '_LS_DB'    ), fbIdList );

stConfig.TimeMax  := F_IDLIST_GETREAL( CONCAT(sHead, '_TimeMax'  ), fbIdList );
stConfig.Delay_Up := F_IDLIST_GETREAL( CONCAT(sHead, '_Delay_Up' ), fbIdList );
stConfig.Delay_Dw := F_IDLIST_GETREAL( CONCAT(sHead, '_Delay_Dw' ), fbIdList );
stConfig.Cycle    := rTime;

stConfig.HP_Up  := F_IDLIST_GETBYTE( CONCAT(sHead, '_HP_Up'  ), fbIdList );
stConfig.HP_Dw  := F_IDLIST_GETBYTE( CONCAT(sHead, '_HP_Dw'  ), fbIdList );
END_FUNCTION

(* POU FUN/PARAMETERS/F_READ_DE_CYLINDER_POS_CFG, ST *)
FUNCTION F_READ_DE_CYLINDER_POS_CFG : BOOL
VAR_INPUT
	sHead : STRING;
	rTime : REAL;
END_VAR
VAR_IN_OUT
	stConfig : ST_DE_CYLINDER_POS_CFG;
	fbIdList : FB_IDLIST;
END_VAR
stConfig.TgtLS_In  := F_IDLIST_GETREAL( CONCAT(sHead, '_TgtLS_In'  ), fbIdList );
stConfig.TgtLS_Out := F_IDLIST_GETREAL( CONCAT(sHead, '_TgtLS_Out' ), fbIdList );
stConfig.TgtLS_Mid := F_IDLIST_GETREAL( CONCAT(sHead, '_TgtLS_Mid' ), fbIdList );
stConfig.TgtLS_DB  := F_IDLIST_GETREAL( CONCAT(sHead, '_TgtLS_DB'  ), fbIdList );

stConfig.TimeMax  := F_IDLIST_GETREAL( CONCAT(sHead, '_TimeMax'  ), fbIdList );
stConfig.Cycle    := rTime;

stConfig.LS_Limit_In  := F_IDLIST_GETBOOL( CONCAT(sHead, '_LS_Limit_In'  ), fbIdList );
stConfig.LS_Limit_Out := F_IDLIST_GETBOOL( CONCAT(sHead, '_LS_Limit_Out' ), fbIdList );

stConfig.HP  := F_IDLIST_GETBYTE( CONCAT(sHead, '_HP'  ), fbIdList );
END_FUNCTION

(* POU FUN/PARAMETERS/F_READ_WB_CFG, ST *)
FUNCTION F_READ_WB_CFG : BOOL
VAR_INPUT
	sHead : STRING;
	rTime : REAL;
END_VAR
VAR_IN_OUT
	stConfig : ST_WB_CFG;
	fbIdList : FB_IDLIST;
END_VAR
VAR
END_VAR
stConfig.Cycle    := rTime;
stConfig.TimeMax_Idle  := F_IDLIST_GETREAL( CONCAT(sHead, '_TimeMax_Idle'   ), fbIdList );
stConfig.TimeMax_Init  := F_IDLIST_GETREAL( CONCAT(sHead, '_TimeMax_Init'   ), fbIdList );
stConfig.TimeMax_DumpFwd  := F_IDLIST_GETREAL( CONCAT(sHead, '_TimeMax_DumpFwd'   ), fbIdList );
stConfig.TimeMax_DumpAft  := F_IDLIST_GETREAL( CONCAT(sHead, '_TimeMax_DumpAft'   ), fbIdList );
stConfig.TimeMax_MoveFwd  := F_IDLIST_GETREAL( CONCAT(sHead, '_TimeMax_MoveFwd'   ), fbIdList );
stConfig.TimeMax_MoveAft  := F_IDLIST_GETREAL( CONCAT(sHead, '_TimeMax_MoveAft'   ), fbIdList );

stConfig.EVP_Pump_Min := F_IDLIST_GETREAL( CONCAT(sHead, '_EVP_Pump_Min' ), fbIdList );
stConfig.EVP_Pump_Max := F_IDLIST_GETREAL( CONCAT(sHead, '_EVP_Pump_Max' ), fbIdList );
stConfig.EVP_Pump_Inc := F_IDLIST_GETREAL( CONCAT(sHead, '_EVP_Pump_Inc' ), fbIdList );
stConfig.EVP_Pump_Dec := F_IDLIST_GETREAL( CONCAT(sHead, '_EVP_Pump_Dec' ), fbIdList );

stConfig.LP := F_IDLIST_GETBYTE( CONCAT(sHead, '_LP' ), fbIdList );

stConfig.EnScoopAF := F_IDLIST_GETBOOL( CONCAT(sHead, '_EnScoopAF' ), fbIdList );
END_FUNCTION

(* POU FUN/PARAMETERS/F_READ_WB_VALVESF_CFG, ST *)
FUNCTION F_READ_WB_VALVESF_CFG : BOOL
VAR_INPUT
	sHead : STRING;
	rTime : REAL;
END_VAR
VAR_IN_OUT
	stConfig : ST_WB_VALVE_CFG;
	fbIdList : FB_IDLIST;
END_VAR
VAR
END_VAR
stConfig.Cycle    := rTime;
stConfig.TimeMax  := F_IDLIST_GETREAL( CONCAT(sHead, '_TimeMax'   ), fbIdList );
stConfig.PushTime := F_IDLIST_GETREAL( CONCAT(sHead, '_PushTime'  ), fbIdList );
stConfig.PushP    := F_IDLIST_GETREAL( CONCAT(sHead, '_PushPress' ), fbIdList );
stConfig.HP       := F_IDLIST_GETBYTE( CONCAT(sHead, '_HP'        ), fbIdList );
END_FUNCTION

(* POU FUN/PARAMETERS/F_READ_WB_VALVELS_CFG, ST *)
FUNCTION F_READ_WB_VALVELS_CFG : BOOL
VAR_INPUT
	sHead : STRING;
	rTime : REAL;
END_VAR
VAR_IN_OUT
	stConfig : ST_WB_VALVE_LS_CFG;
	fbIdList : FB_IDLIST;
END_VAR
VAR
END_VAR
stConfig.Cycle    := rTime;
stConfig.TimeMax  := F_IDLIST_GETREAL( CONCAT(sHead, '_TimeMax'   ), fbIdList );
stConfig.PushTime := F_IDLIST_GETREAL( CONCAT(sHead, '_PushTime'  ), fbIdList );
stConfig.PushP    := F_IDLIST_GETREAL( CONCAT(sHead, '_PushPress' ), fbIdList );

stConfig.TgtLS_Half := F_IDLIST_GETREAL( CONCAT(sHead, '_TgtLS_Half' ), fbIdList );
stConfig.LS_DB      := F_IDLIST_GETREAL( CONCAT(sHead, '_LS_DB'      ), fbIdList );

stConfig.HP := F_IDLIST_GETBYTE( CONCAT(sHead, '_HP' ), fbIdList );
END_FUNCTION

(* POU FUN/PARAMETERS/F_READ_WINCHE_CFG, ST *)
FUNCTION F_READ_WINCHE_CFG : BOOL
VAR_INPUT
	sHead : STRING;
	rTime : REAL;
END_VAR
VAR_IN_OUT
	stConfig : ST_WINCHE_CFG;
	fbIdList : FB_IDLIST;
END_VAR
VAR
	aux1 : REAL;
	aux2 : REAL;
	aux3 : REAL;
END_VAR
stConfig.Spd1[1] := F_IDLIST_GETREAL( CONCAT(sHead, '_Spd11' ), fbIdList );
stConfig.Spd2[1] := F_IDLIST_GETREAL( CONCAT(sHead, '_Spd21' ), fbIdList );
stConfig.Spd3[1] := F_IDLIST_GETREAL( CONCAT(sHead, '_Spd31' ), fbIdList );

stConfig.Spd1[7] := F_IDLIST_GETREAL( CONCAT(sHead, '_Spd17' ), fbIdList );
stConfig.Spd2[7] := F_IDLIST_GETREAL( CONCAT(sHead, '_Spd27' ), fbIdList );
stConfig.Spd3[7] := F_IDLIST_GETREAL( CONCAT(sHead, '_Spd37' ), fbIdList );

stConfig.P1_Max := F_IDLIST_GETREAL( CONCAT(sHead, '_P1_Max' ), fbIdList );
stConfig.P2_Max := F_IDLIST_GETREAL( CONCAT(sHead, '_P2_Max' ), fbIdList );
stConfig.P3_Max := F_IDLIST_GETREAL( CONCAT(sHead, '_P3_Max' ), fbIdList );

stConfig.A_Spd1 := F_IDLIST_GETBOOL( CONCAT(sHead, '_A_Spd1' ), fbIdList );

stConfig.TimeMax := F_IDLIST_GETREAL( CONCAT(sHead, '_TimeMax' ), fbIdList );
stConfig.Cycle   := rTime;

(*stConfig.PP  := F_IDLIST_GETBYTE( CONCAT(sHead, '_PP' ), fbIdList );*)

aux1 := (stConfig.Spd1[7]-stConfig.Spd1[1])/6.0;
aux2 := (stConfig.Spd2[7]-stConfig.Spd2[1])/6.0;
aux3 := (stConfig.Spd3[7]-stConfig.Spd3[1])/6.0;

stConfig.Spd1[2] := stConfig.Spd1[1] + Aux1;
stConfig.Spd1[3] := stConfig.Spd1[2] + Aux1;
stConfig.Spd1[4] := stConfig.Spd1[3] + Aux1;
stConfig.Spd1[5] := stConfig.Spd1[4] + Aux1;
stConfig.Spd1[6] := stConfig.Spd1[5] + Aux1;

stConfig.Spd2[2] := stConfig.Spd2[1] + Aux2;
stConfig.Spd2[3] := stConfig.Spd2[2] + Aux2;
stConfig.Spd2[4] := stConfig.Spd2[3] + Aux2;
stConfig.Spd2[5] := stConfig.Spd2[4] + Aux2;
stConfig.Spd2[6] := stConfig.Spd2[5] + Aux2;

stConfig.Spd3[2] := stConfig.Spd3[1] + Aux3;
stConfig.Spd3[3] := stConfig.Spd3[2] + Aux3;
stConfig.Spd3[4] := stConfig.Spd3[3] + Aux3;
stConfig.Spd3[5] := stConfig.Spd3[4] + Aux3;
stConfig.Spd3[6] := stConfig.Spd3[5] + Aux3;
END_FUNCTION

(* POU FUN/PARAMETERS/F_READ_BOARD_CFG, ST *)
FUNCTION F_READ_BOARD_CFG : BOOL
VAR_INPUT
	sHead : STRING;
	rTime : REAL;
END_VAR
VAR_IN_OUT
	stConfig : ST_BOARD_CFG;
	fbIdList : FB_IDLIST;
END_VAR
VAR
END_VAR
stConfig.TgtLS_P_In   := F_IDLIST_GETREAL( CONCAT(sHead, '_TgtLS_P_In'   ), fbIdList );
stConfig.TgtLS_P_InR  := F_IDLIST_GETREAL( CONCAT(sHead, '_TgtLS_P_InR'  ), fbIdList );
stConfig.TgtLS_P_Out  := F_IDLIST_GETREAL( CONCAT(sHead, '_TgtLS_P_Out'  ), fbIdList );
stConfig.TgtLS_P_OutR := F_IDLIST_GETREAL( CONCAT(sHead, '_TgtLS_P_OutR' ), fbIdList );
stConfig.TgtLS_P_Mid  := F_IDLIST_GETREAL( CONCAT(sHead, '_TgtLS_P_Mid'  ), fbIdList );

stConfig.TgtLS_S_In   := F_IDLIST_GETREAL( CONCAT(sHead, '_TgtLS_S_In'   ), fbIdList );
stConfig.TgtLS_S_InR  := F_IDLIST_GETREAL( CONCAT(sHead, '_TgtLS_S_InR'  ), fbIdList );
stConfig.TgtLS_S_Out  := F_IDLIST_GETREAL( CONCAT(sHead, '_TgtLS_S_Out'  ), fbIdList );
stConfig.TgtLS_S_OutR := F_IDLIST_GETREAL( CONCAT(sHead, '_TgtLS_S_OutR' ), fbIdList );
stConfig.TgtLS_S_Mid  := F_IDLIST_GETREAL( CONCAT(sHead, '_TgtLS_S_Mid'  ), fbIdList );

stConfig.TgtLS_P_Safe_In  := F_IDLIST_GETREAL( CONCAT(sHead, '_TgtLS_P_Safe_In'  ), fbIdList );
stConfig.TgtLS_P_Safe_Out := F_IDLIST_GETREAL( CONCAT(sHead, '_TgtLS_P_Safe_Out' ), fbIdList );

stConfig.TgtLS_S_Safe_In  := F_IDLIST_GETREAL( CONCAT(sHead, '_TgtLS_S_Safe_In'  ), fbIdList );
stConfig.TgtLS_S_Safe_Out := F_IDLIST_GETREAL( CONCAT(sHead, '_TgtLS_S_Safe_Out' ), fbIdList );

stConfig.LS_Dif_Tgt := F_IDLIST_GETREAL( CONCAT(sHead, '_LS_Dif_Tgt' ), fbIdList );
stConfig.LS_Dif_Max := F_IDLIST_GETREAL( CONCAT(sHead, '_LS_Dif_Max' ), fbIdList );
stConfig.LS_Dif_Min := F_IDLIST_GETREAL( CONCAT(sHead, '_LS_Dif_Min' ), fbIdList );

stConfig.LS_DB   := F_IDLIST_GETREAL( CONCAT(sHead, '_LS_DB'   ), fbIdList );

stConfig.P_Hyst_HP := F_IDLIST_GETREAL( CONCAT(sHead, '_P_Hyst_HP' ), fbIdList );
stConfig.P_Hyst_LP := F_IDLIST_GETREAL( CONCAT(sHead, '_P_Hyst_LP' ), fbIdList );
stConfig.P_Hyst_TM := F_IDLIST_GETREAL( CONCAT(sHead, '_P_Hyst_TM' ), fbIdList );

(*Keel Limits*)
stConfig.Keel_P_Max := F_IDLIST_GETREAL( CONCAT(sHead, '_Keel_P_Max' ), fbIdList );
stConfig.Keel_S_Min := F_IDLIST_GETREAL( CONCAT(sHead, '_Keel_S_Min' ), fbIdList );

(*Valve Limits*)
stConfig.EVP_In_P_Min := F_IDLIST_GETREAL( CONCAT(sHead, '_EVP_In_P_Min' ), fbIdList );
stConfig.EVP_In_P_Max := F_IDLIST_GETREAL( CONCAT(sHead, '_EVP_In_P_Max' ), fbIdList );

stConfig.EVP_In_S_Min := F_IDLIST_GETREAL( CONCAT(sHead, '_EVP_In_S_Min' ), fbIdList );
stConfig.EVP_In_S_Max := F_IDLIST_GETREAL( CONCAT(sHead, '_EVP_In_S_Max' ), fbIdList );

stConfig.EVP_Out_P_Min := F_IDLIST_GETREAL( CONCAT(sHead, '_EVP_Out_P_Min' ), fbIdList );
stConfig.EVP_Out_P_Max := F_IDLIST_GETREAL( CONCAT(sHead, '_EVP_Out_P_Max' ), fbIdList );

stConfig.EVP_Out_S_Min := F_IDLIST_GETREAL( CONCAT(sHead, '_EVP_Out_S_Min' ), fbIdList );
stConfig.EVP_Out_S_Max := F_IDLIST_GETREAL( CONCAT(sHead, '_EVP_Out_S_Max' ), fbIdList );

(*Valve Targets*)
stConfig.EVP_In_P_Eng := F_IDLIST_GETREAL( CONCAT(sHead, '_EVP_In_P_Eng' ), fbIdList );
stConfig.EVP_In_P_PP  := F_IDLIST_GETREAL( CONCAT(sHead, '_EVP_In_P_PP'  ), fbIdList );

stConfig.EVP_In_S_Eng := F_IDLIST_GETREAL( CONCAT(sHead, '_EVP_In_S_Eng' ), fbIdList );
stConfig.EVP_In_S_PP  := F_IDLIST_GETREAL( CONCAT(sHead, '_EVP_In_S_PP'  ), fbIdList );

stConfig.EVP_Out_P_Eng := F_IDLIST_GETREAL( CONCAT(sHead, '_EVP_Out_P_Eng' ), fbIdList );
stConfig.EVP_Out_P_PP  := F_IDLIST_GETREAL( CONCAT(sHead, '_EVP_Out_P_PP'  ), fbIdList );

stConfig.EVP_Out_S_Eng := F_IDLIST_GETREAL( CONCAT(sHead, '_EVP_Out_S_Eng' ), fbIdList );
stConfig.EVP_Out_S_PP  := F_IDLIST_GETREAL( CONCAT(sHead, '_EVP_Out_S_PP'  ), fbIdList );

(*Valve Gains*)
stConfig.EVP_In_EVP_K  := F_IDLIST_GETREAL( CONCAT(sHead, '_EVP_In_EVP_K'  ), fbIdList );
stConfig.EVP_Out_EVP_K := F_IDLIST_GETREAL( CONCAT(sHead, '_EVP_Out_EVP_K' ), fbIdList );

stConfig.EVP_In_LS_K  := F_IDLIST_GETREAL( CONCAT(sHead, '_EVP_In_LS_K'  ), fbIdList );
stConfig.EVP_Out_LS_K := F_IDLIST_GETREAL( CONCAT(sHead, '_EVP_Out_LS_K' ), fbIdList );

(*Valve Softstart*)
stConfig.EVP_In_Inc  := F_IDLIST_GETREAL( CONCAT(sHead, '_EVP_In_Inc'  ), fbIdList );
stConfig.EVP_Out_Inc := F_IDLIST_GETREAL( CONCAT(sHead, '_EVP_Out_Inc' ), fbIdList );

stConfig.EVP_In_Dec  := F_IDLIST_GETREAL( CONCAT(sHead, '_EVP_In_Dec'  ), fbIdList );
stConfig.EVP_Out_Dec := F_IDLIST_GETREAL( CONCAT(sHead, '_EVP_Out_Dec' ), fbIdList );

stConfig.LP := F_IDLIST_GETBYTE( CONCAT(sHead, '_LP' ), fbIdList );

stConfig.TimeMax  := F_IDLIST_GETREAL( CONCAT(sHead, '_TimeMax'  ), fbIdList );
stConfig.Cycle    := rTime;
END_FUNCTION

(* POU FUN/PARAMETERS/F_READ_KEEL_CFG, ST *)
FUNCTION F_READ_KEEL_CFG : BOOL
VAR_INPUT
	sHead : STRING;
	rTime : REAL;
END_VAR
VAR_IN_OUT
	stConfig : ST_KEEL_CFG;
	fbIdList : FB_IDLIST;
END_VAR
VAR
END_VAR
(*Targets*)
stConfig.TgtLS_In  := F_IDLIST_GETREAL( CONCAT(sHead, '_TgtLS_In'  ), fbIdList );
stConfig.TgtLS_Mid := F_IDLIST_GETREAL( CONCAT(sHead, '_TgtLS_Mid' ), fbIdList );
stConfig.TgtLS_Out := F_IDLIST_GETREAL( CONCAT(sHead, '_TgtLS_Out' ), fbIdList );

stConfig.TgtLS_Safe_In  := F_IDLIST_GETREAL( CONCAT(sHead, '_TgtLS_Safe_In'  ), fbIdList );
stConfig.TgtLS_Safe_Out := F_IDLIST_GETREAL( CONCAT(sHead, '_TgtLS_Safe_Out' ), fbIdList );

stConfig.TgtLS_Tack_Off := F_IDLIST_GETREAL( CONCAT(sHead, '_TgtLS_Tack_Off' ), fbIdList );

stConfig.LS_DB := F_IDLIST_GETREAL( CONCAT(sHead, '_LS_DB' ), fbIdList );

(*Board Limits*)
stConfig.Board_P_Min_Out := F_IDLIST_GETREAL( CONCAT(sHead, '_Board_P_Min_Out' ), fbIdList );
stConfig.Board_S_Min_Out := F_IDLIST_GETREAL( CONCAT(sHead, '_Board_S_Min_Out' ), fbIdList );

(*Valve Limits*)
stConfig.EVP_In_SE_Min   := F_IDLIST_GETREAL( CONCAT(sHead, '_EVP_In_SE_Min'   ), fbIdList );
stConfig.EVP_In_SE_Max   := F_IDLIST_GETREAL( CONCAT(sHead, '_EVP_In_SE_Max'   ), fbIdList );
stConfig.EVP_In_SE_Man   := F_IDLIST_GETREAL( CONCAT(sHead, '_EVP_In_SE_Man'   ), fbIdList );

stConfig.EVP_In_FE_Min := F_IDLIST_GETREAL( CONCAT(sHead, '_EVP_In_FE_Min' ), fbIdList );
stConfig.EVP_In_FE_Max := F_IDLIST_GETREAL( CONCAT(sHead, '_EVP_In_FE_Max' ), fbIdList );
stConfig.EVP_In_FE_Man := F_IDLIST_GETREAL( CONCAT(sHead, '_EVP_In_FE_Man' ), fbIdList );

stConfig.EVP_In_Eng_Min := F_IDLIST_GETREAL( CONCAT(sHead, '_EVP_In_Eng_Min' ), fbIdList );
stConfig.EVP_In_Eng_Max := F_IDLIST_GETREAL( CONCAT(sHead, '_EVP_In_Eng_Max' ), fbIdList );
stConfig.EVP_In_Eng_Man := F_IDLIST_GETREAL( CONCAT(sHead, '_EVP_In_Eng_Man' ), fbIdList );

stConfig.EVP_In_P_Empty := F_IDLIST_GETREAL( CONCAT(sHead, '_EVP_In_P_Empty' ), fbIdList );

stConfig.EVP_Out_SE_Min := F_IDLIST_GETREAL( CONCAT(sHead, '_EVP_Out_SE_Min' ), fbIdList );
stConfig.EVP_Out_SE_Max := F_IDLIST_GETREAL( CONCAT(sHead, '_EVP_Out_SE_Max' ), fbIdList );
stConfig.EVP_Out_SE_Man := F_IDLIST_GETREAL( CONCAT(sHead, '_EVP_Out_SE_Man' ), fbIdList );
stConfig.EVP_Out_SE_Empty := F_IDLIST_GETREAL( CONCAT(sHead, '_EVP_Out_SE_Empty' ), fbIdList );

stConfig.EVP_Out_FE_Min := F_IDLIST_GETREAL( CONCAT(sHead, '_EVP_Out_FE_Min' ), fbIdList );
stConfig.EVP_Out_FE_Max := F_IDLIST_GETREAL( CONCAT(sHead, '_EVP_Out_FE_Max' ), fbIdList );
stConfig.EVP_Out_FE_Man := F_IDLIST_GETREAL( CONCAT(sHead, '_EVP_Out_FE_Man' ), fbIdList );

stConfig.EVP_Out_Eng_Min := F_IDLIST_GETREAL( CONCAT(sHead, '_EVP_Out_Eng_Min' ), fbIdList );
stConfig.EVP_Out_Eng_Max := F_IDLIST_GETREAL( CONCAT(sHead, '_EVP_Out_Eng_Max' ), fbIdList );
stConfig.EVP_Out_Eng_Man := F_IDLIST_GETREAL( CONCAT(sHead, '_EVP_Out_Eng_Man' ), fbIdList );

stConfig.EVP_Out_Fill_Min := F_IDLIST_GETREAL( CONCAT(sHead, '_EVP_Out_Fill_Min' ), fbIdList );
stConfig.EVP_Out_Fill_Max := F_IDLIST_GETREAL( CONCAT(sHead, '_EVP_Out_Fill_Max' ), fbIdList );

stConfig.EVP_Out_P_Fill := F_IDLIST_GETREAL( CONCAT(sHead, '_EVP_Out_P_Fill' ), fbIdList );

(*Valve Softstart*)
stConfig.EVP_In_SE_Inc := F_IDLIST_GETREAL( CONCAT(sHead, '_EVP_In_SE_Inc' ), fbIdList );
stConfig.EVP_In_SE_Dec := F_IDLIST_GETREAL( CONCAT(sHead, '_EVP_In_SE_Dec' ), fbIdList );

stConfig.EVP_In_FE_Inc := F_IDLIST_GETREAL( CONCAT(sHead, '_EVP_In_FE_Inc' ), fbIdList );
stConfig.EVP_In_FE_Dec := F_IDLIST_GETREAL( CONCAT(sHead, '_EVP_In_FE_Dec' ), fbIdList );

stConfig.EVP_Out_SE_Inc := F_IDLIST_GETREAL( CONCAT(sHead, '_EVP_Out_SE_Inc' ), fbIdList );
stConfig.EVP_Out_SE_Dec := F_IDLIST_GETREAL( CONCAT(sHead, '_EVP_Out_SE_Dec' ), fbIdList );

stConfig.EVP_Out_FE_Inc := F_IDLIST_GETREAL( CONCAT(sHead, '_EVP_Out_FE_Inc' ), fbIdList );
stConfig.EVP_Out_FE_Dec := F_IDLIST_GETREAL( CONCAT(sHead, '_EVP_Out_FE_Dec' ), fbIdList );

stConfig.EVP_In_Eng_Inc := F_IDLIST_GETREAL( CONCAT(sHead, '_EVP_In_Eng_Inc' ), fbIdList );
stConfig.EVP_In_Eng_Dec := F_IDLIST_GETREAL( CONCAT(sHead, '_EVP_In_Eng_Dec' ), fbIdList );

stConfig.EVP_Out_Eng_Inc := F_IDLIST_GETREAL( CONCAT(sHead, '_EVP_Out_Eng_Inc' ), fbIdList );
stConfig.EVP_Out_Eng_Dec := F_IDLIST_GETREAL( CONCAT(sHead, '_EVP_Out_Eng_Dec' ), fbIdList );

(*Valve Gains*)
stConfig.EVP_In_Eng_K  := F_IDLIST_GETREAL( CONCAT(sHead, '_EVP_In_Eng_K'  ), fbIdList );
stConfig.EVP_Out_Eng_K := F_IDLIST_GETREAL( CONCAT(sHead, '_EVP_Out_Eng_K' ), fbIdList );

stConfig.LP  := F_IDLIST_GETBYTE( CONCAT(sHead, '_LP'  ), fbIdList );

stConfig.TimeMax  := F_IDLIST_GETREAL( CONCAT(sHead, '_TimeMax'  ), fbIdList );
stConfig.Cycle    := rTime;

(*Auto Ease limit*)
stConfig.MinLoadSide_Bar   := F_IDLIST_GETREAL( CONCAT(sHead, '_MinLoadSide_Bar'   ), fbIdList );
stConfig.MaxUnloadSide_Bar := F_IDLIST_GETREAL( CONCAT(sHead, '_MaxUnloadSide_Bar' ), fbIdList );
END_FUNCTION

(* POU FUN/PARAMETERS/F_READ_TRAVELLER_CFG, ST *)
FUNCTION F_READ_TRAVELLER_CFG : BOOL
VAR_INPUT
	sHead : STRING;
	rTime : REAL;
END_VAR
VAR_IN_OUT
	stConfig : ST_TRAVELLER_CFG;
	fbIdList : FB_IDLIST;
END_VAR
VAR
END_VAR
stConfig.MaxEVPA := F_IDLIST_GETREAL( CONCAT(sHead, '_MaxEVPA' ), fbIdList );
stConfig.MaxEVPB := F_IDLIST_GETREAL( CONCAT(sHead, '_MaxEVPB' ), fbIdList );
stConfig.MinEVPA := F_IDLIST_GETREAL( CONCAT(sHead, '_MinEVPA' ), fbIdList );
stConfig.MinEVPB := F_IDLIST_GETREAL( CONCAT(sHead, '_MinEVPB' ), fbIdList );

stConfig.Spd_Inc := F_IDLIST_GETREAL( CONCAT(sHead, '_Spd_Inc' ), fbIdList );
stConfig.Spd_Dec := F_IDLIST_GETREAL( CONCAT(sHead, '_Spd_Dec' ), fbIdList );

stConfig.TgtLS_Max  := F_IDLIST_GETREAL( CONCAT(sHead, '_TgtLS_Max'  ), fbIdList );
stConfig.TgtLS_Zero := F_IDLIST_GETREAL( CONCAT(sHead, '_TgtLS_Zero' ), fbIdList );
stConfig.TgtLS_Min  := F_IDLIST_GETREAL( CONCAT(sHead, '_TgtLS_Min'  ), fbIdList );

stConfig.TgtLS_Tack_Off := F_IDLIST_GETREAL( CONCAT(sHead, '_TgtLS_Tack_Off' ), fbIdList );

stConfig.LS_DB    := F_IDLIST_GETREAL( CONCAT(sHead, '_LS_DB'    ), fbIdList );
stConfig.LS_Dist  := F_IDLIST_GETREAL( CONCAT(sHead, '_LS_Dist'  ), fbIdList );
stConfig.LS_Limit := F_IDLIST_GETBOOL( CONCAT(sHead, '_LS_Limit' ), fbIdList );

stConfig.TimeMax  := F_IDLIST_GETREAL( CONCAT(sHead, '_TimeMax'  ), fbIdList );
stConfig.Cycle    := rTime;

stConfig.Hyst_HP := F_IDLIST_GETREAL( CONCAT(sHead, '_Hyst_HP' ), fbIdList );
stConfig.Hyst_LP := F_IDLIST_GETREAL( CONCAT(sHead, '_Hyst_LP' ), fbIdList );
stConfig.Hyst_TM := F_IDLIST_GETREAL( CONCAT(sHead, '_Hyst_TM' ), fbIdList );


stConfig.HP  := F_IDLIST_GETBYTE( CONCAT(sHead, '_HP'  ), fbIdList );
stConfig.LP  := F_IDLIST_GETBYTE( CONCAT(sHead, '_LP'  ), fbIdList );
END_FUNCTION

(* POU FUN/PARAMETERS/F_READ_LP_FUNC_CFG, ST *)
FUNCTION F_READ_LP_FUNC_CFG : BOOL
VAR_INPUT
	sHead : STRING;
	rTime : REAL;
END_VAR
VAR_IN_OUT
	stConfig : ST_LP_FUNC_CFG;
	fbIdList : FB_IDLIST;
END_VAR
VAR
END_VAR
stConfig.SpdA_Min := F_IDLIST_GETREAL( CONCAT(sHead, '_SpdA_Min' ), fbIdList );
stConfig.SpdA_Max := F_IDLIST_GETREAL( CONCAT(sHead, '_SpdA_Max' ), fbIdList );
stConfig.SpdB_Min := F_IDLIST_GETREAL( CONCAT(sHead, '_SpdB_Min' ), fbIdList );
stConfig.SpdB_Max := F_IDLIST_GETREAL( CONCAT(sHead, '_SpdB_Max' ), fbIdList );

stConfig.Spd_Inc := F_IDLIST_GETREAL( CONCAT(sHead, '_Spd_Inc' ), fbIdList );
stConfig.Spd_Dec := F_IDLIST_GETREAL( CONCAT(sHead, '_Spd_Dec' ), fbIdList );

stConfig.A_Spd1 := F_IDLIST_GETBOOL( CONCAT(sHead, '_A_Spd1' ), fbIdList );

stConfig.SF1_Limit := F_IDLIST_GETBOOL( CONCAT(sHead, '_SF1_Limit' ), fbIdList );
stConfig.SF2_Limit := F_IDLIST_GETBOOL( CONCAT(sHead, '_SF2_Limit' ), fbIdList );

stConfig.TimeMax := F_IDLIST_GETREAL( CONCAT(sHead, '_TimeMax' ), fbIdList );
stConfig.Cycle   := rTime;

(*stConfig.PP  := F_IDLIST_GETBYTE( CONCAT(sHead, '_PP' ), fbIdList );*)
END_FUNCTION

(* POU FUN/PARAMETERS/F_READ_TACK_VALVE_CFG, ST *)
FUNCTION F_READ_TACK_VALVE_CFG : BOOL
VAR_INPUT
	sHead : STRING;
	rTime : REAL;
END_VAR
VAR_IN_OUT
	stConfig : ST_TACK_VALVE_CFG;
	fbIdList : FB_IDLIST;
END_VAR
VAR
END_VAR
stConfig.Cycle    := rTime;
stConfig.TimeMax  := F_IDLIST_GETREAL( CONCAT(sHead, '_TimeMax'   ), fbIdList );

stConfig.Hyst_HeelH := F_IDLIST_GETREAL( CONCAT(sHead, '_Hyst_HeelH' ), fbIdList );
stConfig.Hyst_HeelL := F_IDLIST_GETREAL( CONCAT(sHead, '_Hyst_HeelL' ), fbIdList );
stConfig.Hyst_Time  := F_IDLIST_GETREAL( CONCAT(sHead, '_Hyst_Time'  ), fbIdList );
END_FUNCTION

(* POU FUN/PARAMETERS/F_READ_MAST_SETUP_CFG, ST *)
FUNCTION F_READ_MAST_SETUP_CFG : BOOL
VAR_INPUT
	sHead : STRING;
	rTime : REAL;
END_VAR
VAR_IN_OUT
	stTABLE  : ST_MAST_SETUP;
	fbIdList : FB_IDLIST;
END_VAR
VAR
END_VAR
stTABLE.Cycle    := rTime;

stTABLE.aFSY[1,1] := F_IDLIST_GETREAL( CONCAT(sHead, '_FSY_1_1' ), fbIdList );
stTABLE.aFSY[1,2] := F_IDLIST_GETREAL( CONCAT(sHead, '_FSY_1_2' ), fbIdList );
stTABLE.aFSY[1,3] := F_IDLIST_GETREAL( CONCAT(sHead, '_FSY_1_3' ), fbIdList );
stTABLE.aFSY[1,4] := F_IDLIST_GETREAL( CONCAT(sHead, '_FSY_1_4' ), fbIdList );
stTABLE.aFSY[1,5] := F_IDLIST_GETREAL( CONCAT(sHead, '_FSY_1_5' ), fbIdList );
stTABLE.aFSY[1,6] := F_IDLIST_GETREAL( CONCAT(sHead, '_FSY_1_6' ), fbIdList );

stTABLE.aFSY[2,1] := F_IDLIST_GETREAL( CONCAT(sHead, '_FSY_2_1' ), fbIdList );
stTABLE.aFSY[2,2] := F_IDLIST_GETREAL( CONCAT(sHead, '_FSY_2_2' ), fbIdList );
stTABLE.aFSY[2,3] := F_IDLIST_GETREAL( CONCAT(sHead, '_FSY_2_3' ), fbIdList );
stTABLE.aFSY[2,4] := F_IDLIST_GETREAL( CONCAT(sHead, '_FSY_2_4' ), fbIdList );
stTABLE.aFSY[2,5] := F_IDLIST_GETREAL( CONCAT(sHead, '_FSY_2_5' ), fbIdList );
stTABLE.aFSY[2,6] := F_IDLIST_GETREAL( CONCAT(sHead, '_FSY_2_6' ), fbIdList );

stTABLE.aFSY[3,1] := F_IDLIST_GETREAL( CONCAT(sHead, '_FSY_3_1' ), fbIdList );
stTABLE.aFSY[3,2] := F_IDLIST_GETREAL( CONCAT(sHead, '_FSY_3_2' ), fbIdList );
stTABLE.aFSY[3,3] := F_IDLIST_GETREAL( CONCAT(sHead, '_FSY_3_3' ), fbIdList );
stTABLE.aFSY[3,4] := F_IDLIST_GETREAL( CONCAT(sHead, '_FSY_3_4' ), fbIdList );
stTABLE.aFSY[3,5] := F_IDLIST_GETREAL( CONCAT(sHead, '_FSY_3_5' ), fbIdList );
stTABLE.aFSY[3,6] := F_IDLIST_GETREAL( CONCAT(sHead, '_FSY_3_6' ), fbIdList );

stTABLE.aFSY[4,1] := F_IDLIST_GETREAL( CONCAT(sHead, '_FSY_4_1' ), fbIdList );
stTABLE.aFSY[4,2] := F_IDLIST_GETREAL( CONCAT(sHead, '_FSY_4_2' ), fbIdList );
stTABLE.aFSY[4,3] := F_IDLIST_GETREAL( CONCAT(sHead, '_FSY_4_3' ), fbIdList );
stTABLE.aFSY[4,4] := F_IDLIST_GETREAL( CONCAT(sHead, '_FSY_4_4' ), fbIdList );
stTABLE.aFSY[4,5] := F_IDLIST_GETREAL( CONCAT(sHead, '_FSY_4_5' ), fbIdList );
stTABLE.aFSY[4,6] := F_IDLIST_GETREAL( CONCAT(sHead, '_FSY_4_6' ), fbIdList );

stTABLE.aBDef[1,1] := F_IDLIST_GETREAL( CONCAT(sHead, '_BDEF_1_1' ), fbIdList );
stTABLE.aBDef[1,2] := F_IDLIST_GETREAL( CONCAT(sHead, '_BDEF_1_2' ), fbIdList );
stTABLE.aBDef[1,3] := F_IDLIST_GETREAL( CONCAT(sHead, '_BDEF_1_3' ), fbIdList );
stTABLE.aBDef[1,4] := F_IDLIST_GETREAL( CONCAT(sHead, '_BDEF_1_4' ), fbIdList );
stTABLE.aBDef[1,5] := F_IDLIST_GETREAL( CONCAT(sHead, '_BDEF_1_5' ), fbIdList );
stTABLE.aBDef[1,6] := F_IDLIST_GETREAL( CONCAT(sHead, '_BDEF_1_6' ), fbIdList );

stTABLE.aBDef[2,1] := F_IDLIST_GETREAL( CONCAT(sHead, '_BDEF_2_1' ), fbIdList );
stTABLE.aBDef[2,2] := F_IDLIST_GETREAL( CONCAT(sHead, '_BDEF_2_2' ), fbIdList );
stTABLE.aBDef[2,3] := F_IDLIST_GETREAL( CONCAT(sHead, '_BDEF_2_3' ), fbIdList );
stTABLE.aBDef[2,4] := F_IDLIST_GETREAL( CONCAT(sHead, '_BDEF_2_4' ), fbIdList );
stTABLE.aBDef[2,5] := F_IDLIST_GETREAL( CONCAT(sHead, '_BDEF_2_5' ), fbIdList );
stTABLE.aBDef[2,6] := F_IDLIST_GETREAL( CONCAT(sHead, '_BDEF_2_6' ), fbIdList );

stTABLE.aBDef[3,1] := F_IDLIST_GETREAL( CONCAT(sHead, '_BDEF_3_1' ), fbIdList );
stTABLE.aBDef[3,2] := F_IDLIST_GETREAL( CONCAT(sHead, '_BDEF_3_2' ), fbIdList );
stTABLE.aBDef[3,3] := F_IDLIST_GETREAL( CONCAT(sHead, '_BDEF_3_3' ), fbIdList );
stTABLE.aBDef[3,4] := F_IDLIST_GETREAL( CONCAT(sHead, '_BDEF_3_4' ), fbIdList );
stTABLE.aBDef[3,5] := F_IDLIST_GETREAL( CONCAT(sHead, '_BDEF_3_5' ), fbIdList );
stTABLE.aBDef[3,6] := F_IDLIST_GETREAL( CONCAT(sHead, '_BDEF_3_6' ), fbIdList );

stTABLE.aBDef[4,1] := F_IDLIST_GETREAL( CONCAT(sHead, '_BDEF_4_1' ), fbIdList );
stTABLE.aBDef[4,2] := F_IDLIST_GETREAL( CONCAT(sHead, '_BDEF_4_2' ), fbIdList );
stTABLE.aBDef[4,3] := F_IDLIST_GETREAL( CONCAT(sHead, '_BDEF_4_3' ), fbIdList );
stTABLE.aBDef[4,4] := F_IDLIST_GETREAL( CONCAT(sHead, '_BDEF_4_4' ), fbIdList );
stTABLE.aBDef[4,5] := F_IDLIST_GETREAL( CONCAT(sHead, '_BDEF_4_5' ), fbIdList );
stTABLE.aBDef[4,6] := F_IDLIST_GETREAL( CONCAT(sHead, '_BDEF_4_6' ), fbIdList );

stTABLE.aTDef[1,1] := F_IDLIST_GETREAL( CONCAT(sHead, '_TDEF_1_1' ), fbIdList );
stTABLE.aTDef[1,2] := F_IDLIST_GETREAL( CONCAT(sHead, '_TDEF_1_2' ), fbIdList );
stTABLE.aTDef[1,3] := F_IDLIST_GETREAL( CONCAT(sHead, '_TDEF_1_3' ), fbIdList );
stTABLE.aTDef[1,4] := F_IDLIST_GETREAL( CONCAT(sHead, '_TDEF_1_4' ), fbIdList );
stTABLE.aTDef[1,5] := F_IDLIST_GETREAL( CONCAT(sHead, '_TDEF_1_5' ), fbIdList );
stTABLE.aTDef[1,6] := F_IDLIST_GETREAL( CONCAT(sHead, '_TDEF_1_6' ), fbIdList );

stTABLE.aTDef[2,1] := F_IDLIST_GETREAL( CONCAT(sHead, '_TDEF_2_1' ), fbIdList );
stTABLE.aTDef[2,2] := F_IDLIST_GETREAL( CONCAT(sHead, '_TDEF_2_2' ), fbIdList );
stTABLE.aTDef[2,3] := F_IDLIST_GETREAL( CONCAT(sHead, '_TDEF_2_3' ), fbIdList );
stTABLE.aTDef[2,4] := F_IDLIST_GETREAL( CONCAT(sHead, '_TDEF_2_4' ), fbIdList );
stTABLE.aTDef[2,5] := F_IDLIST_GETREAL( CONCAT(sHead, '_TDEF_2_5' ), fbIdList );
stTABLE.aTDef[2,6] := F_IDLIST_GETREAL( CONCAT(sHead, '_TDEF_2_6' ), fbIdList );

stTABLE.aTDef[3,1] := F_IDLIST_GETREAL( CONCAT(sHead, '_TDEF_3_1' ), fbIdList );
stTABLE.aTDef[3,2] := F_IDLIST_GETREAL( CONCAT(sHead, '_TDEF_3_2' ), fbIdList );
stTABLE.aTDef[3,3] := F_IDLIST_GETREAL( CONCAT(sHead, '_TDEF_3_3' ), fbIdList );
stTABLE.aTDef[3,4] := F_IDLIST_GETREAL( CONCAT(sHead, '_TDEF_3_4' ), fbIdList );
stTABLE.aTDef[3,5] := F_IDLIST_GETREAL( CONCAT(sHead, '_TDEF_3_5' ), fbIdList );
stTABLE.aTDef[3,6] := F_IDLIST_GETREAL( CONCAT(sHead, '_TDEF_3_6' ), fbIdList );

stTABLE.aTDef[4,1] := F_IDLIST_GETREAL( CONCAT(sHead, '_TDEF_4_1' ), fbIdList );
stTABLE.aTDef[4,2] := F_IDLIST_GETREAL( CONCAT(sHead, '_TDEF_4_2' ), fbIdList );
stTABLE.aTDef[4,3] := F_IDLIST_GETREAL( CONCAT(sHead, '_TDEF_4_3' ), fbIdList );
stTABLE.aTDef[4,4] := F_IDLIST_GETREAL( CONCAT(sHead, '_TDEF_4_4' ), fbIdList );
stTABLE.aTDef[4,5] := F_IDLIST_GETREAL( CONCAT(sHead, '_TDEF_4_5' ), fbIdList );
stTABLE.aTDef[4,6] := F_IDLIST_GETREAL( CONCAT(sHead, '_TDEF_4_6' ), fbIdList );
END_FUNCTION

(* POU FUN/PARAMETERS/F_WRITE_SENSOR_BAR, ST *)
FUNCTION F_WRITE_SENSOR_BAR : BOOL
VAR_INPUT
	wSize   :DWORD;
	pBuffer :POINTER TO BYTE;
END_VAR
VAR_IN_OUT
	wPos     : DWORD;
	stSensor : ST_SENSOR_BAR;
END_VAR
VAR
END_VAR
F_ADD_STRINGX4_TO_BUFFER( S1:= CONCAT(stSensor.Name, '_K'   ), S2:='$t', S3:= REAL_TO_STRING( stSensor.Cal_K  ), S4:='$n', wSize := wSize, pBuffer := pBuffer, wPos := wPos );
F_ADD_STRINGX4_TO_BUFFER( S1:= CONCAT(stSensor.Name, '_Max' ), S2:='$t', S3:= REAL_TO_STRING( stSensor.MaxBar ), S4:='$n', wSize := wSize, pBuffer := pBuffer, wPos := wPos );
END_FUNCTION

(* POU FUN/PARAMETERS/F_WRITE_SENSOR_TEMP, ST *)
FUNCTION F_WRITE_SENSOR_TEMP : BOOL
VAR_INPUT
	wSize   :DWORD;
	pBuffer :POINTER TO BYTE;
END_VAR
VAR_IN_OUT
	wPos     : DWORD;
	stSensor : ST_SENSOR_TEMP;
END_VAR
VAR
END_VAR
F_ADD_STRINGX4_TO_BUFFER( S1:= CONCAT(stSensor.Name, '_K'   ), S2:='$t', S3:= REAL_TO_STRING( stSensor.Cal_K  ), S4:='$n', wSize := wSize, pBuffer := pBuffer, wPos := wPos );
F_ADD_STRINGX4_TO_BUFFER( S1:= CONCAT(stSensor.Name, '_Off' ), S2:='$t', S3:= REAL_TO_STRING( stSensor.Cal_Off  ), S4:='$n', wSize := wSize, pBuffer := pBuffer, wPos := wPos );

F_ADD_STRINGX4_TO_BUFFER( S1:= CONCAT(stSensor.Name, '_Mild' ), S2:='$t', S3:= REAL_TO_STRING( stSensor.LowDeg ), S4:='$n', wSize := wSize, pBuffer := pBuffer, wPos := wPos );
F_ADD_STRINGX4_TO_BUFFER( S1:= CONCAT(stSensor.Name, '_High' ), S2:='$t', S3:= REAL_TO_STRING( stSensor.HigDeg ), S4:='$n', wSize := wSize, pBuffer := pBuffer, wPos := wPos );
F_ADD_STRINGX4_TO_BUFFER( S1:= CONCAT(stSensor.Name, '_Max'  ), S2:='$t', S3:= REAL_TO_STRING( stSensor.MaxDeg ), S4:='$n', wSize := wSize, pBuffer := pBuffer, wPos := wPos );
F_ADD_STRINGX4_TO_BUFFER( S1:= CONCAT(stSensor.Name, '_Dly'  ), S2:='$t', S3:= REAL_TO_STRING( stSensor.Delay  ), S4:='$n', wSize := wSize, pBuffer := pBuffer, wPos := wPos );
END_FUNCTION

(* POU FUN/PARAMETERS/F_WRITE_SENSOR_POS, ST *)
FUNCTION F_WRITE_SENSOR_POS : BOOL
VAR_INPUT
	wSize   :DWORD;
	pBuffer :POINTER TO BYTE;
END_VAR
VAR_IN_OUT
	wPos     : DWORD;
	stSensor : ST_SENSOR_POS;
END_VAR
VAR
END_VAR
F_ADD_STRINGX4_TO_BUFFER( S1:= CONCAT(stSensor.Name, '_K'   ), S2:='$t', S3:= REAL_TO_STRING( stSensor.Cal_K   ), S4:='$n', wSize := wSize, pBuffer := pBuffer, wPos := wPos );
F_ADD_STRINGX4_TO_BUFFER( S1:= CONCAT(stSensor.Name, '_Off' ), S2:='$t', S3:= REAL_TO_STRING( stSensor.Cal_Off ), S4:='$n', wSize := wSize, pBuffer := pBuffer, wPos := wPos );
END_FUNCTION

(* POU FUN/PARAMETERS/F_WRITE_SENSOR_KG, ST *)
FUNCTION F_WRITE_SENSOR_KG : BOOL
VAR_INPUT
	wSize   :DWORD;
	pBuffer :POINTER TO BYTE;
END_VAR
VAR_IN_OUT
	wPos     : DWORD;
	stSensor : ST_SENSOR_KG;
END_VAR
VAR
END_VAR
F_ADD_STRINGX4_TO_BUFFER( S1:= CONCAT(stSensor.Name, '_K' ), S2:='$t', S3:= REAL_TO_STRING( stSensor.Cal_K ), S4:='$n', wSize := wSize, pBuffer := pBuffer, wPos := wPos );
F_ADD_STRINGX4_TO_BUFFER( S1:= CONCAT(stSensor.Name, '_C' ), S2:='$t', S3:= REAL_TO_STRING( stSensor.Cal_C ), S4:='$n', wSize := wSize, pBuffer := pBuffer, wPos := wPos );
END_FUNCTION

(* POU FUN/PARAMETERS/F_WRITE_ENGINE_CFG, ST *)
FUNCTION F_WRITE_ENGINE_CFG : BOOL
VAR_INPUT
	sHead   : STRING;
	wSize   : DWORD;
	pBuffer : POINTER TO BYTE;
END_VAR
VAR_IN_OUT
	wBufPos     : DWORD;
	stEngineCfg : ST_ENGINE_CFG;
END_VAR
VAR
	fbParamList: BOOL;
END_VAR
F_ADD_STRINGX3_TO_BUFFER( S1:= '$n#', S2:= sHead, S3:=' - Parameters:$n', wSize := wSize, pBuffer := pBuffer, wPos := wBufPos );

F_ADD_STRINGX4_TO_BUFFER( S1:= CONCAT(sHead, '_Min_RPM'   ), S2:='$t', S3:= REAL_TO_STRING( stEngineCfg.Min_RPM    ), S4:='$n', wSize := wSize, pBuffer := pBuffer, wPos := wBufPos );
F_ADD_STRINGX4_TO_BUFFER( S1:= CONCAT(sHead, '_Max_RPM'   ), S2:='$t', S3:= REAL_TO_STRING( stEngineCfg.Max_RPM    ), S4:='$n', wSize := wSize, pBuffer := pBuffer, wPos := wBufPos );
F_ADD_STRINGX4_TO_BUFFER( S1:= CONCAT(sHead, '_Boost_RPM' ), S2:='$t', S3:= REAL_TO_STRING( stEngineCfg.Boost_RPM  ), S4:='$n', wSize := wSize, pBuffer := pBuffer, wPos := wBufPos );
F_ADD_STRINGX4_TO_BUFFER( S1:= CONCAT(sHead, '_Stop_RPM'  ), S2:='$t', S3:= REAL_TO_STRING( stEngineCfg.Stop_RPM   ), S4:='$n', wSize := wSize, pBuffer := pBuffer, wPos := wBufPos );
F_ADD_STRINGX4_TO_BUFFER( S1:= CONCAT(sHead, '_MaxInc_RPM'), S2:='$t', S3:= REAL_TO_STRING( stEngineCfg.MaxInc_RPM ), S4:='$n', wSize := wSize, pBuffer := pBuffer, wPos := wBufPos );
F_ADD_STRINGX4_TO_BUFFER( S1:= CONCAT(sHead, '_MaxDec_RPM'), S2:='$t', S3:= REAL_TO_STRING( stEngineCfg.MaxDec_RPM ), S4:='$n', wSize := wSize, pBuffer := pBuffer, wPos := wBufPos );
F_ADD_STRINGX4_TO_BUFFER( S1:= CONCAT(sHead, '_DlyDec_sec'), S2:='$t', S3:= REAL_TO_STRING( stEngineCfg.DlyDec_sec ), S4:='$n', wSize := wSize, pBuffer := pBuffer, wPos := wBufPos );

F_ADD_STRINGX4_TO_BUFFER( S1:= CONCAT(sHead, '_HP_Nx_RPM'), S2:='$t', S3:= REAL_TO_STRING( stEngineCfg.HP_Nx_RPM ), S4:='$n', wSize := wSize, pBuffer := pBuffer, wPos := wBufPos );
F_ADD_STRINGX4_TO_BUFFER( S1:= CONCAT(sHead, '_HP_SF_RPM'), S2:='$t', S3:= REAL_TO_STRING( stEngineCfg.HP_SF_RPM ), S4:='$n', wSize := wSize, pBuffer := pBuffer, wPos := wBufPos );

F_ADD_STRINGX4_TO_BUFFER( S1:= CONCAT(sHead, '_LP_CK_RPM'), S2:='$t', S3:= REAL_TO_STRING( stEngineCfg.LP_CK_RPM ), S4:='$n', wSize := wSize, pBuffer := pBuffer, wPos := wBufPos );
F_ADD_STRINGX4_TO_BUFFER( S1:= CONCAT(sHead, '_LP_1x_RPM'), S2:='$t', S3:= REAL_TO_STRING( stEngineCfg.LP_1x_RPM ), S4:='$n', wSize := wSize, pBuffer := pBuffer, wPos := wBufPos );
F_ADD_STRINGX4_TO_BUFFER( S1:= CONCAT(sHead, '_LP_2x_RPM'), S2:='$t', S3:= REAL_TO_STRING( stEngineCfg.LP_2x_RPM ), S4:='$n', wSize := wSize, pBuffer := pBuffer, wPos := wBufPos );
F_ADD_STRINGX4_TO_BUFFER( S1:= CONCAT(sHead, '_LP_3x_RPM'), S2:='$t', S3:= REAL_TO_STRING( stEngineCfg.LP_3x_RPM ), S4:='$n', wSize := wSize, pBuffer := pBuffer, wPos := wBufPos );
F_ADD_STRINGX4_TO_BUFFER( S1:= CONCAT(sHead, '_LP_Nx_RPM'), S2:='$t', S3:= REAL_TO_STRING( stEngineCfg.LP_Nx_RPM ), S4:='$n', wSize := wSize, pBuffer := pBuffer, wPos := wBufPos );

F_ADD_STRINGX4_TO_BUFFER( S1:= CONCAT(sHead, '_N_WinchWOP'), S2:='$t', S3:= INT_TO_STRING( stEngineCfg.N_Winch_WOP ), S4:='$n', wSize := wSize, pBuffer := pBuffer, wPos := wBufPos );
F_ADD_STRINGX4_TO_BUFFER( S1:= CONCAT(sHead, '_N_WinchWK' ), S2:='$t', S3:= INT_TO_STRING( stEngineCfg.N_Winch_WK  ), S4:='$n', wSize := wSize, pBuffer := pBuffer, wPos := wBufPos );
F_ADD_STRINGX4_TO_BUFFER( S1:= CONCAT(sHead, '_N_WinchWP' ), S2:='$t', S3:= INT_TO_STRING( stEngineCfg.N_Winch_WP  ), S4:='$n', wSize := wSize, pBuffer := pBuffer, wPos := wBufPos );

F_ADD_STRINGX4_TO_BUFFER( S1:= CONCAT(sHead, '_Max_Torque'), S2:='$t', S3:= REAL_TO_STRING( stEngineCfg.Max_Torque ), S4:='$n', wSize := wSize, pBuffer := pBuffer, wPos := wBufPos );
F_ADD_STRINGX4_TO_BUFFER( S1:= CONCAT(sHead, '_Min_Torque'), S2:='$t', S3:= REAL_TO_STRING( stEngineCfg.Min_Torque ), S4:='$n', wSize := wSize, pBuffer := pBuffer, wPos := wBufPos );

F_ADD_STRINGX4_TO_BUFFER( S1:= CONCAT(sHead, '_Inc_RMP_Perc_WOP'), S2:='$t', S3:= REAL_TO_STRING( stEngineCfg.Inc_RMP_Perc_WOP ), S4:='$n', wSize := wSize, pBuffer := pBuffer, wPos := wBufPos );
F_ADD_STRINGX4_TO_BUFFER( S1:= CONCAT(sHead, '_Dec_Flow_Perc_WP'), S2:='$t', S3:= REAL_TO_STRING( stEngineCfg.Dec_Flow_Perc_WP ), S4:='$n', wSize := wSize, pBuffer := pBuffer, wPos := wBufPos );

F_ADD_STRINGX4_TO_BUFFER( S1:= CONCAT(sHead, '_Max_HeatExch_P'), S2:='$t', S3:= REAL_TO_STRING( stEngineCfg.Max_HeatExch_P ), S4:='$n', wSize := wSize, pBuffer := pBuffer, wPos := wBufPos );

F_ADD_STRINGX4_TO_BUFFER( S1:= CONCAT(sHead, '_EnForceRPM'), S2:='$t', S3:= BOOL_TO_STRING( stEngineCfg.EnForceRPM ), S4:='$n', wSize := wSize, pBuffer := pBuffer, wPos := wBufPos );
F_ADD_STRINGX4_TO_BUFFER( S1:= CONCAT(sHead, '_EnForceTHR'), S2:='$t', S3:= BOOL_TO_STRING( stEngineCfg.EnForceTHR ), S4:='$n', wSize := wSize, pBuffer := pBuffer, wPos := wBufPos );
END_FUNCTION

(* POU FUN/PARAMETERS/F_WRITE_POWERPACK_CFG, ST *)
FUNCTION F_WRITE_POWERPACK_CFG : BOOL
VAR_INPUT
	sHead : STRING;
	wSize   :DWORD;
	pBuffer :POINTER TO BYTE;
END_VAR
VAR_IN_OUT
	wPos     : DWORD;
	stConfig : ST_POWERPACK_CFG;
END_VAR
VAR
END_VAR
F_ADD_STRINGX3_TO_BUFFER( S1:= '$n#', S2:= sHead, S3:=' - Parameters:$n', wSize := wSize, pBuffer := pBuffer, wPos := wPos );

F_ADD_STRINGX4_TO_BUFFER( S1:= CONCAT(sHead, '_Hyst_HP' ), S2:='$t', S3:= REAL_TO_STRING( stConfig.Hyst_HP ), S4:='$n', wSize := wSize, pBuffer := pBuffer, wPos := wPos );
F_ADD_STRINGX4_TO_BUFFER( S1:= CONCAT(sHead, '_Hyst_LP' ), S2:='$t', S3:= REAL_TO_STRING( stConfig.Hyst_LP ), S4:='$n', wSize := wSize, pBuffer := pBuffer, wPos := wPos );
F_ADD_STRINGX4_TO_BUFFER( S1:= CONCAT(sHead, '_Hyst_TM' ), S2:='$t', S3:= REAL_TO_STRING( stConfig.Hyst_TM ), S4:='$n', wSize := wSize, pBuffer := pBuffer, wPos := wPos );

F_ADD_STRINGX4_TO_BUFFER( S1:= CONCAT(sHead, '_Thr_HP' ), S2:='$t', S3:= REAL_TO_STRING( stConfig.Thr_HP ), S4:='$n', wSize := wSize, pBuffer := pBuffer, wPos := wPos );
F_ADD_STRINGX4_TO_BUFFER( S1:= CONCAT(sHead, '_Thr_LP' ), S2:='$t', S3:= REAL_TO_STRING( stConfig.Thr_LP ), S4:='$n', wSize := wSize, pBuffer := pBuffer, wPos := wPos );
END_FUNCTION

(* POU FUN/PARAMETERS/F_WRITE_PROPULSION_CFG, ST *)
FUNCTION F_WRITE_PROPULSION_CFG : BOOL
VAR_INPUT
	sHead : STRING;
	wSize   :DWORD;
	pBuffer :POINTER TO BYTE;
END_VAR
VAR_IN_OUT
	wBufPos         : DWORD;
	stPropulsionCfg : ST_PROPULSION_CFG;
END_VAR
VAR
END_VAR
F_ADD_STRINGX3_TO_BUFFER( S1:= '$n#', S2:= sHead, S3:=' - Parameters:$n', wSize := wSize, pBuffer := pBuffer, wPos := wBufPos );

F_ADD_STRINGX4_TO_BUFFER( S1:= CONCAT(sHead, '_Thrt0_V' ), S2:='$t', S3:= REAL_TO_STRING( stPropulsionCfg.aThrt_V[0]  ), S4:='$n', wSize := wSize, pBuffer := pBuffer, wPos := wBufPos );
F_ADD_STRINGX4_TO_BUFFER( S1:= CONCAT(sHead, '_Thrt4_V' ), S2:='$t', S3:= REAL_TO_STRING( stPropulsionCfg.aThrt_V[4]  ), S4:='$n', wSize := wSize, pBuffer := pBuffer, wPos := wBufPos );
F_ADD_STRINGX4_TO_BUFFER( S1:= CONCAT(sHead, '_Thrt5_V' ), S2:='$t', S3:= REAL_TO_STRING( stPropulsionCfg.aThrt_V[5]  ), S4:='$n', wSize := wSize, pBuffer := pBuffer, wPos := wBufPos );
F_ADD_STRINGX4_TO_BUFFER( S1:= CONCAT(sHead, '_Thrt6_V' ), S2:='$t', S3:= REAL_TO_STRING( stPropulsionCfg.aThrt_V[6]  ), S4:='$n', wSize := wSize, pBuffer := pBuffer, wPos := wBufPos );
F_ADD_STRINGX4_TO_BUFFER( S1:= CONCAT(sHead, '_Thrt10_V'), S2:='$t', S3:= REAL_TO_STRING( stPropulsionCfg.aThrt_V[10] ), S4:='$n', wSize := wSize, pBuffer := pBuffer, wPos := wBufPos );
F_ADD_STRINGX4_TO_BUFFER( S1:= CONCAT(sHead, '_ThrDB_V' ), S2:='$t', S3:= REAL_TO_STRING( stPropulsionCfg.IdleDB_V    ), S4:='$n', wSize := wSize, pBuffer := pBuffer, wPos := wBufPos );

F_ADD_STRINGX4_TO_BUFFER( S1:= CONCAT(sHead, '_RPM_K'    ), S2:='$t', S3:= REAL_TO_STRING( stPropulsionCfg.PropRPM_K ), S4:='$n', wSize := wSize, pBuffer := pBuffer, wPos := wBufPos );
F_ADD_STRINGX4_TO_BUFFER( S1:= CONCAT(sHead, '_Delay_Off'), S2:='$t', S3:= REAL_TO_STRING( stPropulsionCfg.Delay_Off ), S4:='$n', wSize := wSize, pBuffer := pBuffer, wPos := wBufPos );


F_ADD_STRINGX4_TO_BUFFER( S1:= CONCAT(sHead, '_RPM0' ), S2:='$t', S3:= REAL_TO_STRING( stPropulsionCfg.aEng_RPM[0]  ), S4:='$n', wSize := wSize, pBuffer := pBuffer, wPos := wBufPos );
F_ADD_STRINGX4_TO_BUFFER( S1:= CONCAT(sHead, '_RPM1' ), S2:='$t', S3:= REAL_TO_STRING( stPropulsionCfg.aEng_RPM[1]  ), S4:='$n', wSize := wSize, pBuffer := pBuffer, wPos := wBufPos );
F_ADD_STRINGX4_TO_BUFFER( S1:= CONCAT(sHead, '_RPM2' ), S2:='$t', S3:= REAL_TO_STRING( stPropulsionCfg.aEng_RPM[2]  ), S4:='$n', wSize := wSize, pBuffer := pBuffer, wPos := wBufPos );
F_ADD_STRINGX4_TO_BUFFER( S1:= CONCAT(sHead, '_RPM3' ), S2:='$t', S3:= REAL_TO_STRING( stPropulsionCfg.aEng_RPM[3]  ), S4:='$n', wSize := wSize, pBuffer := pBuffer, wPos := wBufPos );
F_ADD_STRINGX4_TO_BUFFER( S1:= CONCAT(sHead, '_RPM4' ), S2:='$t', S3:= REAL_TO_STRING( stPropulsionCfg.aEng_RPM[4]  ), S4:='$n', wSize := wSize, pBuffer := pBuffer, wPos := wBufPos );
F_ADD_STRINGX4_TO_BUFFER( S1:= CONCAT(sHead, '_RPM5' ), S2:='$t', S3:= REAL_TO_STRING( 0.0                          ), S4:='$n', wSize := wSize, pBuffer := pBuffer, wPos := wBufPos );
F_ADD_STRINGX4_TO_BUFFER( S1:= CONCAT(sHead, '_RPM6' ), S2:='$t', S3:= REAL_TO_STRING( stPropulsionCfg.aEng_RPM[6]  ), S4:='$n', wSize := wSize, pBuffer := pBuffer, wPos := wBufPos );
F_ADD_STRINGX4_TO_BUFFER( S1:= CONCAT(sHead, '_RPM7' ), S2:='$t', S3:= REAL_TO_STRING( stPropulsionCfg.aEng_RPM[7]  ), S4:='$n', wSize := wSize, pBuffer := pBuffer, wPos := wBufPos );
F_ADD_STRINGX4_TO_BUFFER( S1:= CONCAT(sHead, '_RPM8' ), S2:='$t', S3:= REAL_TO_STRING( stPropulsionCfg.aEng_RPM[8]  ), S4:='$n', wSize := wSize, pBuffer := pBuffer, wPos := wBufPos );
F_ADD_STRINGX4_TO_BUFFER( S1:= CONCAT(sHead, '_RPM9' ), S2:='$t', S3:= REAL_TO_STRING( stPropulsionCfg.aEng_RPM[9]  ), S4:='$n', wSize := wSize, pBuffer := pBuffer, wPos := wBufPos );
F_ADD_STRINGX4_TO_BUFFER( S1:= CONCAT(sHead, '_RPM10'), S2:='$t', S3:= REAL_TO_STRING( stPropulsionCfg.aEng_RPM[10] ), S4:='$n', wSize := wSize, pBuffer := pBuffer, wPos := wBufPos );

